F_BACnetRM_IsErrorSet:=TRUE;
IF stResult^.errorType = E_BACnet_ErrorType.eTypeAbort AND stResult^.abortReason = E_BACnet_AbortReason.eNoError THEN
	F_BACnetRM_IsErrorSet:=FALSE;
	RETURN;
END_IF
IF stResult^.errorType = E_BACnet_ErrorType.eTypeError AND stResult^.errorClass = E_BACnet_ErrorClass.eErrorClassNoError THEN
	F_BACnetRM_IsErrorSet:=FALSE;
	RETURN;
END_IF
IF stResult^.errorType = E_BACnet_ErrorType.eTypeReject AND stResult^.rejectCode = E_BACnet_RejectReason.eNoError THEN
	F_BACnetRM_IsErrorSet:=FALSE;
	RETURN;
END_IF

END_FUNCTION

// POUs/Helper/[internal]/String/F_BACnet_ChrStrExtLen
{attribute 'hide'} // [Workaround] Not hidden when lib is included
FUNCTION INTERNAL F_BACnet_ChrStrExtLen : UDINT
VAR
	pByte	: POINTER TO BYTE;
	nLen	: UDINT;
END_VAR
(*All VAR_IN_OUT variables have been moved to the end of the declaration due to compatibility reasons*)
VAR_IN_OUT
	stCharStringExt	: ST_BACnet_CharacterStringExt;
END_VAR

pByte := ADR(stCharStringExt);
nLen := SIZEOF(stCharStringExt);
(* check the string type *)
IF (nLen > 4 AND stCharStringExt.cookie = 0) THEN
	(* character string ext. *)
	IF (stCharStringExt.strLen <= SIZEOF(stCharStringExt.stringData)) THEN
		(* plausible string length given *)
		F_BACnet_ChrStrExtLen := stCharStringExt.strLen;
		RETURN;
	END_IF
	(* use sizeof, because string length isn't plausible *)
	nLen := SIZEOF(stCharStringExt.stringData);
	(* re-adjust pointer *)
	pByte := ADR(stCharStringExt.stringData);
END_IF
(* scan zero termination *)
F_BACnet_ChrStrExtLen := 0;
WHILE ((pByte^ <> 0) AND (F_BACnet_ChrStrExtLen < nLen)) DO
	pByte := pByte + 1;
	F_BACnet_ChrStrExtLen := F_BACnet_ChrStrExtLen + 1;
END_WHILE

END_FUNCTION

// POUs/Helper/[internal]/String/F_BACnet_DecodeUCS2
{attribute 'hide'} // [Workaround] Not hidden when lib is included
FUNCTION INTERNAL F_BACnet_DecodeUCS2 : UDINT (* result is the new character length of the string *)
VAR_INPUT
	pString		: POINTER TO WORD; (* pointer to UCS2 string beginning *)
	nString	: UDINT; (* byte size of string (use SIZEOF - don't use LEN) *)
END_VAR
VAR
	i		: UDINT;
	pResult	: POINTER TO BYTE;
	pBy		: POINTER TO WORD;
END_VAR

pResult	:= pString;
pBy		:= pString;
FOR i := 0 TO nString-1 DO
	pResult^ := F_BACnet_UCS2ToWin1252(pBy, TRUE);
	pBy := pBy + 2;
	(* end-of-string by character *)
	IF (pResult^ = 16#00) THEN
		EXIT;
	END_IF
	(* next character *)
	pResult := pResult + 1;
	(* end-of-string by length *)
	IF (pBy >= (pString + nString)) THEN
		EXIT;
	END_IF
END_FOR
pResult^ := 16#00;
F_BACnet_DecodeUCS2 := pResult - pString;

END_FUNCTION

// POUs/Helper/[internal]/String/F_BACnet_UCS2ToWin1252
{attribute 'hide'} // [Workaround] Not hidden when lib is included
FUNCTION INTERNAL F_BACnet_UCS2ToWin1252 : BYTE
VAR_INPUT
	pUCS2 :	POINTER TO WORD;
	bBE	: BOOL; (* byte-order big endian = TRUE *)
END_VAR
VAR
	pArr : POINTER TO ARRAY[0..1] OF BYTE;
	wUCS2: WORD;
END_VAR
VAR CONSTANT
	cRepl	: BYTE := 16#5F;
END_VAR

(*
	Windows-Codepages
874		Thai
932		Japanisch
936		Vereinfachtes Chinesisch
949		Koreanisch
950		Traditionelles Chinesisch
1250	Mitteleuropäisch
1251	Kyrillisch
1252	Westeuropäisch
1253	Griechisch
1254	Türkisch
1255	Hebräisch
1256	Arabisch
1257	Baltisch
1258	Vietnamesisch
*)
pArr := pUCS2;
IF bBE THEN
	wUCS2 := (pArr^[0] * 16#0100) + pArr^[1];
ELSE
	wUCS2 := pUCS2^;
END_IF
CASE wUCS2 OF
	16#178: 	F_BACnet_UCS2ToWin1252 := 16#9F;
	16#153: 	F_BACnet_UCS2ToWin1252 := 16#9C;
	16#152: 	F_BACnet_UCS2ToWin1252 := 16#8C;
	16#17E: 	F_BACnet_UCS2ToWin1252 := 16#9E;
	16#17D: 	F_BACnet_UCS2ToWin1252 := 16#8E;
	16#161: 	F_BACnet_UCS2ToWin1252 := 16#9A;
	16#160: 	F_BACnet_UCS2ToWin1252 := 16#8A;
	16#20AC: 	F_BACnet_UCS2ToWin1252 := 16#80;
	ELSE
		IF wUCS2 <= 16#FF THEN
			F_BACnet_UCS2ToWin1252 := WORD_TO_BYTE(wUCS2);
		ELSE
			F_BACnet_UCS2ToWin1252 := cRepl;
		END_IF
END_CASE

END_FUNCTION

// POUs/Helper/[internal]/String/F_BACnet_DecodeUCS4
{attribute 'hide'} // [Workaround] Not hidden when lib is included
FUNCTION INTERNAL F_BACnet_DecodeUCS4 : UDINT (* result is the new character length of the string *)
VAR_INPUT
	pString		: POINTER TO DWORD; (* pointer to UCS4 string beginning *)
	nString	: UDINT; (* byte size of string (use SIZEOF - don't use LEN) *)
END_VAR
VAR
	i		: UDINT;
	pResult	: POINTER TO BYTE;
	pBy		: POINTER TO WORD;
END_VAR

pResult	:= pString;
pBy		:= pString;
FOR i := 0 TO nString-1 DO
	(* byte order big endian *)
	pResult^ := F_BACnet_UCS2ToWin1252(pBy+2, TRUE);
	pBy := pBy + 4;
	(* end-of-string by character *)
	IF (pResult^ = 16#00) THEN
		EXIT;
	END_IF
	(* next character *)
	pResult := pResult + 1;
	(* end-of-string by length *)
	IF (pBy >= (pString + nString)) THEN
		EXIT;
	END_IF
END_FOR
pResult^ := 16#00;
F_BACnet_DecodeUCS4 := pResult - pString;

END_FUNCTION

// POUs/Helper/[internal]/String/F_BACnet_DecodeUTF8
{attribute 'hide'} // [Workaround] Not hidden when lib is included
FUNCTION INTERNAL F_BACnet_DecodeUTF8 : UDINT (* result is the new character length of the string *)
VAR_INPUT
	pString		: POINTER TO BYTE; (* pointer to UTF-8 string beginning *)
	nString	: UDINT; (* byte size of string (use SIZEOF - don't use LEN) *)
END_VAR
VAR
	i			: UDINT;
	pResult		: POINTER TO BYTE;
	pBy			: POINTER TO BYTE;
	pByArr		: POINTER TO ARRAY[0..3] OF BYTE;
END_VAR

pResult	:= pString;
pBy		:= pString;
FOR i := 0 TO nString-1 DO
	pByArr := pBy;
	IF (pByArr^[0] AND 16#F0) = 16#C0 THEN
		IF (pByArr^[1] AND 16#80) = 16#80 THEN
			pResult^ := F_BACnet_Utf8ToWin1252(pByArr, 2);
			pBy := pBy + 2;
		END_IF
	ELSIF (pByArr^[0] AND 16#F0) = 16#E0 THEN
		IF (pByArr^[1] AND 16#80) = 16#80 THEN
			IF (pByArr^[2] AND 16#80) = 16#80 THEN
				pResult^ := F_BACnet_Utf8ToWin1252(pByArr, 3);
				pBy := pBy + 3;
			END_IF
		END_IF
	ELSIF (pByArr^[0] AND 16#F0) = 16#F0 THEN
		IF (pByArr^[1] AND 16#80) = 16#80 THEN
			IF (pByArr^[2] AND 16#80) = 16#80 THEN
				IF (pByArr^[3] AND 16#80) = 16#80 THEN
					pResult^ := F_BACnet_Utf8ToWin1252(pByArr, 4);
					pBy := pBy + 4;
				END_IF
			END_IF
		END_IF
	ELSE
		(* ASCII character *)
		pResult^ := pBy^;
		pBy := pBy + 1;
	END_IF
	(* end-of-string by character *)
	IF (pResult^ = 16#00) THEN
		EXIT;
	END_IF
	(* next character *)
	pResult := pResult + 1;
	(* end-of-string by length *)
	IF (pBy >= (pString + nString)) THEN
		EXIT;
	END_IF
END_FOR
pResult^ := 16#00;
F_BACnet_DecodeUTF8 := pResult - pString;

END_FUNCTION

// POUs/Helper/[internal]/String/F_BACnet_Utf8ToWin1252
{attribute 'hide'} // [Workaround] Not hidden when lib is included
FUNCTION INTERNAL F_BACnet_Utf8ToWin1252 : BYTE
VAR_INPUT
	pUtf8	: POINTER TO BYTE;
	nUtf8	: UDINT; (* byte size of UTF8 character (1...6) *)
END_VAR
VAR
	pArr		: POINTER TO ARRAY[0..5] OF BYTE;
	pWord		: POINTER TO ARRAY[0..1] OF BYTE;
	wUCS2		: WORD;
END_VAR
VAR CONSTANT
	cRepl	: BYTE := 16#5F;
END_VAR

(*
	Windows-Codepages
874		Thai
932		Japanisch
936		Vereinfachtes Chinesisch
949		Koreanisch
950		Traditionelles Chinesisch
1250	Mitteleuropäisch
1251	Kyrillisch
1252	Westeuropäisch
1253	Griechisch
1254	Türkisch
1255	Hebräisch
1256	Arabisch
1257	Baltisch
1258	Vietnamesisch
*)
(* first step - convert to UCS2 *)
pArr := pUtf8;
IF (pArr^[0] <= 16#7F) THEN
	(* basic latin *)
	F_BACnet_Utf8ToWin1252 := pArr^[0];
	RETURN;
ELSIF (nUtf8 >= 2) THEN
	pWord := ADR(wUCS2);
	IF (pArr^[0] = 16#C2) THEN
		(* latin-1 supplement *)
		wUCS2 := pArr^[1];
	ELSIF (pArr^[0] = 16#C3) AND (pArr^[1] <= 16#BF) THEN
		(* latin-1 supplement *)
		wUCS2 := pArr^[1] + 16#40;
	ELSIF (pArr^[0] = 16#C4) AND (pArr^[1] >= 16#80) THEN
		(* latin extended-A *)
		pWord^[1] := 16#01;
		pWord^[0] := pArr^[1] - 16#80;
	ELSIF (pArr^[0] = 16#C5) AND (pArr^[1] >= 16#80) THEN
		(* latin extended-A *)
		pWord^[1] := 16#01;
		pWord^[0] := pArr^[1] - 16#40;
	ELSIF (pArr^[0] = 16#C6) AND (pArr^[1] >= 16#80) THEN
		(* latin extended-B *)
		pWord^[1] := 16#01;
		pWord^[0] := pArr^[1];
	ELSIF (pArr^[0] = 16#C7) AND (pArr^[1] <= 16#BF) THEN
		(* latin extended-B *)
		pWord^[1] := 16#01;
		pWord^[0] := pArr^[1] + 16#40;
	ELSIF (nUtf8 >= 3) THEN
		IF (pArr^[0] = 16#E2) AND (pArr^[1] = 16#82) THEN
			(* currency symbols *)
			pWord^[1] := 16#20;
			pWord^[0] := pArr^[2];
		ELSE
			(* unsupported *)
			F_BACnet_Utf8ToWin1252 := cRepl;
			RETURN;
		END_IF
	ELSE
		(* unsupported *)
		F_BACnet_Utf8ToWin1252 := cRepl;
		RETURN;
	END_IF
	(* convert UCS2 to Windows-1252 *)
	F_BACnet_Utf8ToWin1252 := F_BACnet_UCS2ToWin1252(pWord, FALSE);
	RETURN;
END_IF
(* unsupported *)
F_BACnet_Utf8ToWin1252 := cRepl;

END_FUNCTION

// POUs/Helper/[internal]/String/F_BACnet_EncodeUTF8
{attribute 'hide'} // [Workaround] Not hidden when lib is included
FUNCTION INTERNAL F_BACnet_EncodeUTF8 : UDINT (* actually byte length of the result utf-8 string (maybe longer than cbResult; means overflow) *)
VAR_INPUT
	pString		: POINTER TO BYTE; (* pointer to Win1252 string beginning *)
	nString	: UDINT; (* byte size of string (use SIZEOF - don't use LEN) *)
	pResult		: POINTER TO BYTE; (* pointer to result UTF-8 data area *)
	nResult	: UDINT; (* byte size of result (use SIZEOF - don't use LEN) *)
END_VAR

VAR
	pBy			: POINTER TO BYTE;
	pByArr		: POINTER TO ARRAY[0..3] OF BYTE;
	nCoded		: UINT;
	bOverflow	: BOOL;
END_VAR
(*All VAR_IN_OUT variables have been moved to the end of the declaration due to compatibility reasons*)
VAR_IN_OUT
	nResultLen	: UDINT; (* final resulting string length (<= nResult) *)
END_VAR

pBy			:= pString;
pByArr		:= pResult;
bOverflow	:= FALSE;
F_BACnet_EncodeUTF8 := 0;
nResultLen	:= 0;
(* loop over pString *)
WHILE pBy < (pString + nString) DO
	IF (pBy^ = 0) THEN EXIT; END_IF
	IF bOverflow OR (F_BACnet_EncodeUTF8 + 3 > nResult) THEN
		nCoded := F_BACnet_Win1252ToUtf8(nW1252:=pBy^, pUtf8:=pByArr, bEval:=TRUE);
		IF (NOT bOverflow) AND (F_BACnet_EncodeUTF8 + nCoded <= nResult) THEN
			nCoded := F_BACnet_Win1252ToUtf8(nW1252:=pBy^, pUtf8:=pByArr, bEval:=FALSE);
		ELSE
			bOverflow := TRUE;
		END_IF
	ELSE
		nCoded := F_BACnet_Win1252ToUtf8(nW1252:=pBy^, pUtf8:=pByArr, bEval:=FALSE);
	END_IF
	IF (NOT bOverflow) THEN
		pByArr := pByArr + UINT_TO_UDINT(nCoded);
		nResultLen := F_BACnet_EncodeUTF8 + nCoded;
	END_IF
	F_BACnet_EncodeUTF8 := F_BACnet_EncodeUTF8 + nCoded;
	pBy := pBy + 1;
END_WHILE
(* add zero termination if needed *)
IF (nResultLen < nResult) THEN
	pByArr^[0] := 16#00;
END_IF

END_FUNCTION

// POUs/Helper/[internal]/String/F_BACnet_Win1252ToUtf8
{attribute 'hide'} // [Workaround] Not hidden when lib is included
FUNCTION INTERNAL F_BACnet_Win1252ToUtf8 : UINT(0..3)
VAR_INPUT
	nW1252	: BYTE; (* Win1252 character *)
	pUtf8	: POINTER TO ARRAY[0..2] OF BYTE; (* pointer to target character buffer (utf-8) *)
	bEval	: BOOL; (* TRUE = only evaluate expected coding size (0..3 byte) - but don't write data *)
END_VAR
VAR
	pWord	: POINTER TO ARRAY[0..1] OF BYTE;
	wUCS2	: WORD;
END_VAR
VAR CONSTANT
	cRepl	: BYTE := 16#5F;
END_VAR

(*
	Windows-Codepages
874		Thai
932		Japanisch
936		Vereinfachtes Chinesisch
949		Koreanisch
950		Traditionelles Chinesisch
1250	Mitteleuropäisch
1251	Kyrillisch
1252	Westeuropäisch
1253	Griechisch
1254	Türkisch
1255	Hebräisch
1256	Arabisch
1257	Baltisch
1258	Vietnamesisch
*)
(* check pointer *)
IF (pUtf8 = 0) THEN
	(* null pointer *)
	F_BACnet_Win1252ToUtf8 := 0;
ELSIF (nW1252 <= 16#7F) THEN
	(* basic latin - 1 byte *)
	IF (NOT bEval) THEN
		pUtf8^[0] := nW1252;
	END_IF
	F_BACnet_Win1252ToUtf8 := 1;
ELSE
	(* convert to UCS-2 first *)
	wUCS2 := F_BACnet_Win1252ToUCS2(nW1252:=nW1252, bBE:=FALSE);
	pWord := ADR(wUCS2);
	(* convert used ranges *)
	IF (wUCS2 >= 16#80 AND wUCS2 <= 16#BF) THEN
		(* latin-1 supplement *)
		IF (NOT bEval) THEN
			pUtf8^[0] := 16#C2;
			pUtf8^[1] := pWord^[0];
		END_IF
		F_BACnet_Win1252ToUtf8 := 2;
	ELSIF (wUCS2 >= 16#C0 AND wUCS2 <= 16#FF) THEN
		(* latin-1 supplement *)
		IF (NOT bEval) THEN
			pUtf8^[0] := 16#C3;
			pUtf8^[1] := pWord^[0] - 16#40;
		END_IF
		F_BACnet_Win1252ToUtf8 := 2;
	ELSIF (wUCS2 >= 16#140 AND wUCS2 <= 16#17F) THEN
		(* latin extended A *)
		IF (NOT bEval) THEN
			pUtf8^[0] := 16#C5;
			pUtf8^[1] := pWord^[0] + 16#40;
		END_IF
		F_BACnet_Win1252ToUtf8 := 2;
	ELSIF (wUCS2 >= 16#20A0 AND wUCS2 <= 16#20BF) THEN
		(* currency symbols *)
		IF (NOT bEval) THEN
			pUtf8^[0] := 16#E2;
			pUtf8^[1] := 16#82;
			pUtf8^[2] := pWord^[0];
		END_IF
		F_BACnet_Win1252ToUtf8 := 3;
	ELSE
		(* unsupported *)
		IF (NOT bEval) THEN
			pUtf8^[0] := cRepl;
		END_IF
		F_BACnet_Win1252ToUtf8 := 1;
	END_IF
END_IF

END_FUNCTION

// POUs/Helper/[internal]/String/F_BACnet_Win1252ToUCS2
{attribute 'hide'} // [Workaround] Not hidden when lib is included
FUNCTION INTERNAL F_BACnet_Win1252ToUCS2 : WORD
VAR_INPUT
	nW1252 : BYTE;
	bBE	: BOOL; (* byte-order big endian = TRUE *)
END_VAR
VAR
	pArr : POINTER TO ARRAY[0..1] OF BYTE;
	nBuf : BYTE;
	wUCS2: WORD;
END_VAR

(*
	Windows-Codepages
874		Thai
932		Japanisch
936		Vereinfachtes Chinesisch
949		Koreanisch
950		Traditionelles Chinesisch
1250	Mitteleuropäisch
1251	Kyrillisch
1252	Westeuropäisch
1253	Griechisch
1254	Türkisch
1255	Hebräisch
1256	Arabisch
1257	Baltisch
1258	Vietnamesisch
*)
CASE nW1252 OF
	16#9F: wUCS2 := 16#178;
	16#9C: wUCS2 := 16#153;
	16#8C: wUCS2 := 16#152;
	16#9E: wUCS2 := 16#17E;
	16#8E: wUCS2 := 16#17D;
	16#9A: wUCS2 := 16#161;
	16#8A: wUCS2 := 16#160;
	16#80: wUCS2 := 16#20AC;
	ELSE
	wUCS2 := nW1252;
END_CASE
IF bBE THEN
	pArr := ADR(wUCS2);
	nBuf := pArr^[0];
	pArr^[0] := pArr^[1];
	pArr^[1] := nBuf;
END_IF
F_BACnet_Win1252ToUCS2 := wUCS2;

END_FUNCTION

// POUs/Helper/[internal]/String/F_BACnet_GetUsedStateText
{attribute 'hide'} // [Workaround] Not hidden when lib is included
FUNCTION INTERNAL F_BACnet_GetUsedStateText : UDINT
VAR_IN_OUT
	sArray				: ARRAY[*] OF T_BACnet_StateText;
END_VAR
VAR
	_nTemp				: DINT;
END_VAR

F_BACnet_GetUsedStateText := 0;

FOR _nTemp := LOWER_BOUND(sArray, 1) TO UPPER_BOUND(sArray, 1) DO
	IF LEN(sArray[_nTemp]) = 0 THEN
		EXIT;
	ELSE
		F_BACnet_GetUsedStateText := (F_BACnet_GetUsedStateText+1);
	END_IF
END_FOR

END_FUNCTION

// POUs/Helper/[internal]/String/F_BACnet_GetUsedUDINT
{attribute 'hide'} // [Workaround] Not hidden when lib is included
FUNCTION INTERNAL F_BACnet_GetUsedUDINT : UDINT
VAR_IN_OUT
	nArray				: ARRAY[*] OF UDINT;
END_VAR
VAR
	_nTemp				: DINT;
END_VAR

F_BACnet_GetUsedUDINT := 0;

FOR _nTemp := LOWER_BOUND(nArray, 1) TO UPPER_BOUND(nArray, 1) DO
	IF (nArray[_nTemp] = 0) THEN
		EXIT;
	ELSE
		F_BACnet_GetUsedUDINT := (F_BACnet_GetUsedUDINT+1);
	END_IF
END_FOR

END_FUNCTION

// POUs/Helper/[internal]/Validation-Functions/F_BACnet_IsObjIdentifierValid
{attribute 'hide'} // [Workaround] Not hidden when lib is included
FUNCTION INTERNAL F_BACnet_IsObjIdentifierValid : BOOL
VAR_INPUT
	tIdentifier		: T_BACnet_ObjectIdentifier;
END_VAR

F_BACnet_IsObjIdentifierValid := ((tIdentifier <> 0) AND (tIdentifier <> BACnet_Globals.nBACnetObjId_None));

END_FUNCTION

// POUs/Helper/[internal]/Validation-Functions/F_BACnet_IsPriorityValid
{attribute 'hide'} // [Workaround] Not hidden when lib is included
FUNCTION INTERNAL F_BACnet_IsPriorityValid : BOOL
VAR_INPUT
	ePriority		: E_BACnet_Priority;
END_VAR

F_BACnet_IsPriorityValid := ((E_BACnet_Priority.First <= ePriority) AND (ePriority <= E_BACnet_Priority.Last));

END_FUNCTION

// POUs/Helper/[internal]/Validation-Functions/F_BACnet_IsSchedBTypeValid
{attribute 'hide'} // [Workaround] Not hidden when lib is included
FUNCTION INTERNAL F_BACnet_IsSchedBTypeValid : BOOL
VAR_INPUT
	eType		: E_BACnet_SchedBType;
END_VAR

F_BACnet_IsSchedBTypeValid := ((E_BACnet_SchedBType.First <= eType) AND (eType <= E_BACnet_SchedBType.Last));

END_FUNCTION

// POUs/Helper/[internal]/F_BACnet_AlignedSize
{attribute 'hide'} // [Workaround] Not hidden when lib is included
FUNCTION INTERNAL F_BACnet_AlignedSize : DWORD
VAR_INPUT
	n	: DWORD;
END_VAR
VAR
END_VAR

F_BACnet_AlignedSize := (4*(((n)+3)/4));

END_FUNCTION

// POUs/Helper/[internal]/F_BACnet_AnalogPV
{attribute 'hide'} // [Workaround] Not hidden when lib is included
FUNCTION INTERNAL F_BACnet_AnalogPV : REAL
VAR_INPUT
	bEnable	: BOOL; (* TRUE = commit to stack, FALSE = do-nothing *)
	bNull	: BOOL; (* TRUE = clear priority, FALSE = write value from input *)
	fValue	: REAL;
END_VAR
VAR
	pres : POINTER TO DWORD;
END_VAR

IF (bEnable) THEN
	IF (bNull) THEN
		pres := ADR(F_BACnet_AnalogPV);
		pres^ := F_BACnet_RealNull(); 
	ELSE
		F_BACnet_AnalogPV := fValue;
	END_IF
ELSE
	F_BACnet_AnalogPV := F_BACnet_NAN();
END_IF

END_FUNCTION

// POUs/Helper/Real/F_BACnet_RealNull
FUNCTION F_BACnet_RealNull : DWORD
(* function that generates <not-a-number> real state *)

F_BACnet_RealNull:=16#7FFF0000;

END_FUNCTION

// POUs/Helper/Real/F_BACnet_NAN
FUNCTION F_BACnet_NAN : REAL
(* function that generates <not-a-number> real state *)
VAR
	res : POINTER TO DWORD;
END_VAR

res:=ADR(F_BACnet_NAN);
res^:=16#7FFFFFFF;

END_FUNCTION

// POUs/Helper/[internal]/F_BACnet_BitFieldBit
{attribute 'hide'} // [Workaround] Not hidden when lib is included
FUNCTION INTERNAL F_BACnet_BitFieldBit : WORD
VAR_INPUT
	bitNbr	:	INT;
END_VAR
VAR
END_VAR

F_BACnet_BitFieldBit := to_word((bitNbr/8) * 8 + (bitNbr MOD 8));

END_FUNCTION

// POUs/Helper/[internal]/F_BACnet_ChangeBitFieldBit
{attribute 'hide'} // [Workaround] Not hidden when lib is included
FUNCTION INTERNAL F_BACnet_ChangeBitFieldBit : DWORD
VAR_INPUT
	ptrData		: POINTER TO DWORD;
	bitNbr			: INT;
	Value		: BOOL;
END_VAR
VAR
END_VAR

IF (NOT Value) THEN
	ptrData^ := ptrData^ AND NOT (SHR(DWORD#16#00008000,F_BACnet_BitFieldBit(bitNbr)));
ELSE
	ptrData^ := ptrData^ OR (SHR(DWORD#16#00008000,F_BACnet_BitFieldBit(bitNbr)));
END_IF
F_BACnet_ChangeBitFieldBit := ptrData^;

END_FUNCTION

// POUs/Helper/[internal]/F_BACnet_EndOf
{attribute 'hide'} // [Workaround] Not hidden when lib is included
FUNCTION INTERNAL F_BACnet_EndOf : POINTER TO BYTE
VAR_INPUT
	 pPtr : POINTER TO BYTE;
	 nSize : DWORD;
END_VAR
VAR
END_VAR

F_BACnet_EndOf:=pPtr+nSize;

END_FUNCTION

// POUs/Helper/[internal]/F_BACnet_IsBitFieldBitSet
{attribute 'hide'} // [Workaround] Not hidden when lib is included
FUNCTION INTERNAL F_BACnet_IsBitFieldBitSet : BOOL
VAR_INPUT
	data	:	DWORD;
	bitNbr		:	INT;
END_VAR
VAR
END_VAR

F_BACnet_IsBitFieldBitSet:= (data AND (SHR(DWORD#16#00008000,F_BACnet_BitFieldBit(bitNbr)))) > 0;

END_FUNCTION

// POUs/Helper/[internal]/F_BACnet_IsBitFieldBitSetPtr
{attribute 'hide'} // [Workaround] Not hidden when lib is included
FUNCTION INTERNAL F_BACnet_IsBitFieldBitSetPtr : BOOL
VAR_INPUT
	pData	:	POINTER TO WORD;
	bitNbr	:	INT;
END_VAR
VAR
END_VAR

F_BACnet_IsBitFieldBitSetPtr:= ((pData^) AND (SHR(16#8000,F_BACnet_BitFieldBit(bitNbr)))) > 0;

END_FUNCTION

// POUs/Helper/[internal]/F_BACnet_NextListElem
{attribute 'hide'} // [Workaround] Not hidden when lib is included
FUNCTION INTERNAL F_BACnet_NextListElem : POINTER TO BYTE
VAR_INPUT
	 pPtr : POINTER TO BYTE;
	 nSize : DWORD;
END_VAR
VAR
END_VAR

IF nSize < 16#80000000 THEN
	F_BACnet_NextListElem:=0;
	RETURN;
END_IF
F_BACnet_NextListElem:=pPtr+F_BACnet_AlignedSize(nSize AND 16#7FFFFFFF)+8;

END_FUNCTION

// POUs/Helper/[internal]/F_BACnet_SetBitFieldBit
{attribute 'hide'} // [Workaround] Not hidden when lib is included
FUNCTION INTERNAL F_BACnet_SetBitFieldBit : DWORD
VAR_INPUT
	ptrData		:	POINTER TO DWORD;
	bitNbr			:	INT;
END_VAR
VAR
END_VAR

ptrData^ := ptrData^ OR (SHR(DWORD#16#00008000, F_BACnet_BitFieldBit(bitNbr)));
F_BACnet_SetBitFieldBit := ptrData^;

END_FUNCTION

// POUs/Helper/[internal]/F_BACnet_SysTimeDiff
{attribute 'hide'} // [Workaround] Not hidden when lib is included
FUNCTION INTERNAL F_BACnet_SysTimeDiff : REAL
VAR_INPUT
	In1, In2 : T_LARGE_INTEGER;
END_VAR

F_BACnet_SysTimeDiff := LREAL_TO_REAL(INT64_TO_LREAL(Int64Sub64(In1, In2)) / 10000000.0); (* [s] *)

END_FUNCTION

// POUs/Helper/[internal]/F_BACnet_UnSetBitFieldBit
{attribute 'hide'} // [Workaround] Not hidden when lib is included
FUNCTION INTERNAL F_BACnet_UnSetBitFieldBit : DWORD
VAR_INPUT
	ptrData		:	POINTER TO DWORD;
	bitNbr			:	INT;
END_VAR
VAR
END_VAR

ptrData^ := ptrData^ AND NOT (SHR(DWORD#16#00008000,F_BACnet_BitFieldBit(bitNbr)));
F_BACnet_UnSetBitFieldBit := ptrData^;

END_FUNCTION

// POUs/Helper/Flags/F_BACnet_EventEnable
FUNCTION F_BACnet_EventEnable : UINT
VAR_INPUT
	stEvtEn       : ST_BA_EventTransitions;
END_VAR
VAR
	nEvtEnToFlt     : UINT;
	nEvtEnToNmal    : UINT;
	nEvtEnToOffnmal : UINT;
	nEvtEnNo        : UINT;
END_VAR

(*=============================================*)
(*EventEnable*)
IF	stEvtEn.bToFault
THEN
	nEvtEnToFlt := 16#4000;
ELSE
	nEvtEnToFlt := 16#0;
END_IF

IF	stEvtEn.bToNormal
THEN
	nEvtEnToNmal := 16#2000;
ELSE
	nEvtEnToNmal := 16#0;
END_IF

IF	stEvtEn.bToOffnormal
THEN
	nEvtEnToOffnmal := 16#8000;
ELSE
	nEvtEnToOffnmal := 16#0;
END_IF

nEvtEnNo := 5;

F_BACnet_EventEnable := nEvtEnNo + nEvtEnToFlt + nEvtEnToNmal + nEvtEnToOffnmal;
(*=============================================*)

END_FUNCTION

// POUs/Helper/Flags/F_BACnet_EventTransitionFlags
FUNCTION F_BACnet_EventTransitionFlags : ST_BA_EventTransitions
VAR_INPUT
	data	: WORD;
END_VAR
VAR
END_VAR

F_BACnet_EventTransitionFlags.bToNormal := F_BACnet_IsBitFieldBitSet(data, E_BACnet_EventTransitionBits.eToNormal);
F_BACnet_EventTransitionFlags.bToOffnormal := F_BACnet_IsBitFieldBitSet(data, E_BACnet_EventTransitionBits.eToOffnormal);
F_BACnet_EventTransitionFlags.bToFault := F_BACnet_IsBitFieldBitSet(data, E_BACnet_EventTransitionBits.eToFault);

END_FUNCTION

// POUs/Helper/Flags/F_BACnet_GetEventTransFlagsData
FUNCTION F_BACnet_GetEventTransFlagsData : WORD
VAR_INPUT
	Flags	: ST_BA_EventTransitions;
END_VAR
VAR
END_VAR

F_BACnet_GetEventTransFlagsData := 16#0005;
IF Flags.bToNormal THEN
	F_BACnet_GetEventTransFlagsData := DWORD_TO_WORD(F_BACnet_SetBitFieldBit(ptrData:=ADR(F_BACnet_GetEventTransFlagsData), bitNbr:=E_BACnet_EventTransitionBits.eToNormal));
END_IF
IF Flags.bToOffnormal THEN
	F_BACnet_GetEventTransFlagsData := DWORD_TO_WORD(F_BACnet_SetBitFieldBit(ptrData:=ADR(F_BACnet_GetEventTransFlagsData), bitNbr:=E_BACnet_EventTransitionBits.eToOffnormal));
END_IF
IF Flags.bToFault THEN
	F_BACnet_GetEventTransFlagsData := DWORD_TO_WORD(F_BACnet_SetBitFieldBit(ptrData:=ADR(F_BACnet_GetEventTransFlagsData), bitNbr:=E_BACnet_EventTransitionBits.eToFault));
END_IF

END_FUNCTION

// POUs/Helper/Flags/F_BACnet_GetLimitEnFlagsData
FUNCTION F_BACnet_GetLimitEnFlagsData : WORD
VAR_INPUT
	Flags	: ST_BACnet_LimitEnable;
END_VAR
VAR
END_VAR

F_BACnet_GetLimitEnFlagsData := 16#0006;
IF Flags.highLimitEnable THEN
	F_BACnet_GetLimitEnFlagsData := DWORD_TO_WORD(F_BACnet_SetBitFieldBit(ptrData:=ADR(F_BACnet_GetLimitEnFlagsData), bitNbr:=E_BACnet_LimitEnableBits.eHighLimit));
END_IF
IF Flags.lowLimitEnable THEN
	F_BACnet_GetLimitEnFlagsData := DWORD_TO_WORD(F_BACnet_SetBitFieldBit(ptrData:=ADR(F_BACnet_GetLimitEnFlagsData), bitNbr:=E_BACnet_LimitEnableBits.eLowLimit));
END_IF

END_FUNCTION

// POUs/Helper/Flags/F_BACnet_GetStatusFlagsData
FUNCTION F_BACnet_GetStatusFlagsData : WORD
VAR_INPUT
	Flags : ST_BA_StatusFlags;
END_VAR

F_BACnet_GetStatusFlagsData	:= 16#0004;
IF Flags.bInAlarm THEN
	F_BACnet_GetStatusFlagsData := DWORD_TO_WORD(F_BACnet_SetBitFieldBit(ptrData:=ADR(F_BACnet_GetStatusFlagsData), bitNbr:=E_BACnet_StatusFlags.eInAlarm));
END_IF
IF Flags.bFault THEN
	F_BACnet_GetStatusFlagsData := DWORD_TO_WORD(F_BACnet_SetBitFieldBit(ptrData:=ADR(F_BACnet_GetStatusFlagsData), bitNbr:=E_BACnet_StatusFlags.eFault));
END_IF
IF Flags.bOverridden THEN
	F_BACnet_GetStatusFlagsData := DWORD_TO_WORD(F_BACnet_SetBitFieldBit(ptrData:=ADR(F_BACnet_GetStatusFlagsData), bitNbr:=E_BACnet_StatusFlags.eOverridden));
END_IF
IF Flags.bOutOfService THEN
	F_BACnet_GetStatusFlagsData := DWORD_TO_WORD(F_BACnet_SetBitFieldBit(ptrData:=ADR(F_BACnet_GetStatusFlagsData), bitNbr:=E_BACnet_StatusFlags.eOutOfService));
END_IF

END_FUNCTION

// POUs/Helper/Flags/F_BACnet_LimitEnable
FUNCTION F_BACnet_LimitEnable : UINT
VAR_INPUT
	stLimEn         : ST_BACnet_LimitEnable;
END_VAR
VAR
	nHiLimEn     : UINT;
	nLowLimEn    : UINT;
	nLimEnNo     : UINT;
END_VAR

(*=============================================*)
IF	stLimEn.highLimitEnable
THEN
	nHiLimEn := 16#4000;
ELSE
	nHiLimEn := 16#0;
END_IF


IF	stLimEn.lowLimitEnable
THEN
	nLowLimEn := 16#8000;
ELSE
	nLowLimEn := 16#0;
END_IF

nLimEnNo := 16#6;

F_BACnet_LimitEnable := nLimEnNo + nHiLimEn + nLowLimEn;
(*=============================================*)

END_FUNCTION

// POUs/Helper/Flags/F_BACnet_LimitEnableFlags
FUNCTION F_BACnet_LimitEnableFlags : ST_BACnet_LimitEnable
VAR_INPUT
	data	: WORD;
END_VAR
VAR
END_VAR

F_BACnet_LimitEnableFlags.highLimitEnable := F_BACnet_IsBitFieldBitSet( data:=data, bitNbr:=E_BACnet_LimitEnableBits.eHighLimit);
F_BACnet_LimitEnableFlags.lowLimitEnable := F_BACnet_IsBitFieldBitSet( data:=data, bitNbr:=E_BACnet_LimitEnableBits.eLowLimit);

END_FUNCTION

// POUs/Helper/Flags/F_BACnet_StatusFlags
FUNCTION F_BACnet_StatusFlags : ST_BA_StatusFlags
VAR_INPUT
	data	: WORD;
END_VAR
VAR
END_VAR

F_BACnet_StatusFlags.bInAlarm:= F_BACnet_IsBitFieldBitSet( data:=data, bitNbr:=E_BACnet_StatusFlags.eInAlarm);
F_BACnet_StatusFlags.bFault:= F_BACnet_IsBitFieldBitSet( data:=data, bitNbr:=E_BACnet_StatusFlags.eFault);
F_BACnet_StatusFlags.bOverridden:= F_BACnet_IsBitFieldBitSet( data:=data, bitNbr:=E_BACnet_StatusFlags.eOverridden);
F_BACnet_StatusFlags.bOutOfService:= F_BACnet_IsBitFieldBitSet( data:=data, bitNbr:=E_BACnet_StatusFlags.eOutOfService);

END_FUNCTION

// POUs/Helper/MultiState/F_BACnet_EnMultiStatePV
FUNCTION F_BACnet_EnMultiStatePV : UDINT
VAR_INPUT
	bEnable			: BOOL;
	nValue			: UDINT;
END_VAR

IF (bEnable) THEN
	F_BACnet_EnMultiStatePV := MAX(nValue, E_BACnet_MultistateVal.eMin);
ELSE
	F_BACnet_EnMultiStatePV := E_BACnet_MultistateVal.eNull;
END_IF

END_FUNCTION

// POUs/Helper/MultiState/F_BACnet_MultiStatePV
FUNCTION F_BACnet_MultiStatePV : UDINT
VAR_INPUT
	bEnable						: BOOL; (* TRUE = commit to stack, FALSE = do-nothing *)
	bNull						: BOOL; (* TRUE = clear priority, FALSE = write number from state input *)
	nState						: UDINT; (* multi-state [1..max-number-of-states] *)
END_VAR

IF (bEnable) THEN
	IF (bNull) THEN
		F_BACnet_MultiStatePV := E_BACnet_MultistateVal.eNull;
	ELSE
		F_BACnet_MultiStatePV := MAX(nState, E_BACnet_MultistateVal.eMin);
	END_IF
ELSE
	F_BACnet_MultiStatePV := E_BACnet_MultistateVal.eNothing;
END_IF

END_FUNCTION

// POUs/Helper/NC/F_BACnet_DeviceRecipient
// Returns an initialized recipient structure.
FUNCTION F_BACnet_DeviceRecipient : ST_BACnet_Recipient
VAR_INPUT
	nDeviceInstance		: UDINT			:= 16#003FFFFF;
END_VAR

F_BACnet_DeviceRecipient.eRecipientChoice := E_BACnet_RecipientChoice.eDevice;
F_BACnet_DeviceRecipient.stEntry.nDeviceInstance := F_BACnet_GetObjId(E_BACnetObjType.ObjDevice,nDeviceInstance);

END_FUNCTION

// POUs/Helper/F_BACnet_GetObjId
FUNCTION F_BACnet_GetObjId : T_BACnet_ObjectIdentifier
VAR_INPUT
	eObjectType		: E_BACnetObjType;
	nObjectInstance	: UDINT;
END_VAR
VAR
END_VAR

F_BACnet_GetObjId := F_BACnet_GetObjInstance(nObjectInstance) + SHL(INT_TO_UDINT(eObjectType), 22);

END_FUNCTION

// POUs/Helper/F_BACnet_GetObjInstance
FUNCTION F_BACnet_GetObjInstance : UDINT
VAR_INPUT
	nObjectId : DWORD;
END_VAR
VAR
END_VAR

F_BACnet_GetObjInstance := nObjectId AND 16#003FFFFF;

END_FUNCTION

// POUs/Helper/NC/F_BACnet_EthernetRecipient
// Returns an initialized recipient structure.
FUNCTION F_BACnet_EthernetRecipient : ST_BACnet_Recipient
VAR_INPUT
	nIPAddress1		: BYTE;
	nIPAddress2		: BYTE;
	nIPAddress3		: BYTE;
	nIPAddress4		: BYTE;
	nPort			: UINT;
	nNetworkNr		: UINT;
END_VAR
VAR
	_nPort			: POINTER TO ARRAY[0 .. 1] OF BYTE := ADR(nPort);
END_VAR

F_BACnet_EthernetRecipient.eRecipientChoice := E_BACnet_RecipientChoice.eAddress;
F_BACnet_EthernetRecipient.stEntry.stNetAddr.eChoice := E_BACnet_AddressChoice.eEthernet;
F_BACnet_EthernetRecipient.stEntry.stNetAddr.nNetworkNr := nNetworkNr;
F_BACnet_EthernetRecipient.stEntry.stNetAddr.eAddress[0] := nIPAddress1;
F_BACnet_EthernetRecipient.stEntry.stNetAddr.eAddress[1] := nIPAddress2;
F_BACnet_EthernetRecipient.stEntry.stNetAddr.eAddress[2] := nIPAddress3;
F_BACnet_EthernetRecipient.stEntry.stNetAddr.eAddress[3] := nIPAddress4;

// Swap Port-Bytes:
F_BACnet_EthernetRecipient.stEntry.stNetAddr.eAddress[4] := _nPort^[1];
F_BACnet_EthernetRecipient.stEntry.stNetAddr.eAddress[5] := _nPort^[0];

END_FUNCTION

// POUs/Helper/NC/F_BACnet_EthernetRecipientEx
// Returns an initialized recipient structure.
FUNCTION F_BACnet_EthernetRecipientEx : ST_BACnet_Recipient
VAR_INPUT
	tIPAddress		: T_IPv4AddrArr;
	nPort			: UINT;
	nNetworkNr		: UINT;
END_VAR

F_BACnet_EthernetRecipientEx := F_BACnet_EthernetRecipient(tIPAddress[0], tIPAddress[1], tIPAddress[2], tIPAddress[3], nPort, nNetworkNr);

END_FUNCTION

// POUs/Helper/Real/F_BACnet_EnRealPV
FUNCTION F_BACnet_EnRealPV : DWORD
VAR_INPUT
	bEnable	: BOOL;
	fValue	: REAL;
END_VAR
VAR
	pDword : POINTER TO DWORD;
END_VAR

IF (bEnable) THEN
	pDword := ADR(fValue);
	F_BACnet_EnRealPV := pDword^;
ELSE
	F_BACnet_EnRealPV := F_BACnet_RealNull();
END_IF

END_FUNCTION

// POUs/Helper/Real/F_BACnet_IsFinite
FUNCTION F_BACnet_IsFinite : BOOL
VAR_INPUT
	fValue		: REAL;
END_VAR
VAR
	fArg		: T_Arg;
END_VAR

fArg.cbLen := SIZEOF(fValue);
fArg.eType := ARGTYPE_REAL;
fArg.pData := ADR(fValue);
F_BACnet_IsFinite := IsFinite(fArg);

END_FUNCTION

// POUs/Helper/Real/F_BACnet_RealEQ
FUNCTION F_BACnet_RealEQ : BOOL
VAR_INPUT
	fIn1	: REAL;
	fIn2	: REAL;
END_VAR
VAR
END_VAR

IF (F_BACnet_IsFinite(fIn1) <> F_BACnet_IsFinite(fIn2)) THEN
	F_BACnet_RealEQ := FALSE;
	RETURN;
END_IF
IF F_BACnet_IsFinite(fIn1) THEN
	IF (fIn1 <> fIn2) THEN
		F_BACnet_RealEQ := FALSE;
		RETURN;
	END_IF
END_IF
F_BACnet_RealEQ := TRUE;

END_FUNCTION

// POUs/Helper/Real/F_BACnet_RealGE
FUNCTION F_BACnet_RealGE : BOOL
VAR_INPUT
	fIn1	: REAL;
	fIn2	: REAL;
END_VAR
VAR
END_VAR

IF NOT (F_BACnet_IsFinite(fIn1) OR F_BACnet_IsFinite(fIn2)) THEN
	F_BACnet_RealGE := FALSE;
	RETURN;
END_IF
F_BACnet_RealGE := (fIn1 >= fIn2);

END_FUNCTION

// POUs/Helper/Real/F_BACnet_RealGT
FUNCTION F_BACnet_RealGT : BOOL
VAR_INPUT
	fIn1	: REAL;
	fIn2	: REAL;
END_VAR
VAR
END_VAR

IF NOT (F_BACnet_IsFinite(fIn1) OR F_BACnet_IsFinite(fIn2)) THEN
	F_BACnet_RealGT := FALSE;
	RETURN;
END_IF
F_BACnet_RealGT := (fIn1 > fIn2);

END_FUNCTION

// POUs/Helper/Real/F_BACnet_RealLE
FUNCTION F_BACnet_RealLE : BOOL
VAR_INPUT
	fIn1	: REAL;
	fIn2	: REAL;
END_VAR
VAR
END_VAR

IF NOT (F_BACnet_IsFinite(fIn1) OR F_BACnet_IsFinite(fIn2)) THEN
	F_BACnet_RealLE := FALSE;
	RETURN;
END_IF
F_BACnet_RealLE := (fIn1 <= fIn2);

END_FUNCTION

// POUs/Helper/Real/F_BACnet_RealLT
FUNCTION F_BACnet_RealLT : BOOL
VAR_INPUT
	fIn1	: REAL;
	fIn2	: REAL;
END_VAR
VAR
END_VAR

IF NOT (F_BACnet_IsFinite(fIn1) OR F_BACnet_IsFinite(fIn2)) THEN
	F_BACnet_RealLT := FALSE;
	RETURN;
END_IF
F_BACnet_RealLT := (fIn1 < fIn2);

END_FUNCTION

// POUs/Helper/Real/F_BACnet_RealNothing
FUNCTION F_BACnet_RealNothing : DWORD

F_BACnet_RealNothing:=16#7FFFFFFF;

END_FUNCTION

// POUs/Helper/Real/F_BACnet_RealPV
FUNCTION F_BACnet_RealPV : DWORD
VAR_INPUT
	bEnable	: BOOL; (* TRUE = commit to stack, FALSE = do-nothing *)
	bNull	: BOOL; (* TRUE = clear priority, FALSE = write value from input *)
	fValue	: REAL;
END_VAR
VAR
	pDword : POINTER TO DWORD;
END_VAR

IF (bEnable) THEN
	IF (bNull) THEN
		F_BACnet_RealPV := F_BACnet_RealNull();
	ELSE
		pDword := ADR(fValue);
		F_BACnet_RealPV := pDword^;
	END_IF
ELSE
	F_BACnet_RealPV := F_BACnet_RealNothing();
END_IF

END_FUNCTION

// POUs/Helper/Real/F_BACnet_RealToStr
FUNCTION F_BACnet_RealToStr : STRING
VAR_INPUT
	pValue	: POINTER TO REAL;
END_VAR
VAR
	fArg	: T_Arg;
	pDWORD	: POINTER TO DWORD;
END_VAR

IF (pValue <> 0) THEN
	fArg.cbLen := 4;
	fArg.eType := ARGTYPE_REAL;
	fArg.pData := pValue;
	pDWORD := pValue;
	IF IsFinite(fArg) THEN
		F_BACnet_RealToStr := REAL_TO_STRING(pValue^);
	ELSE
		IF (pDWORD^ = 16#7FFF0000) THEN
			F_BACnet_RealToStr := '#NULL';
		ELSIF (pDWORD^ AND 16#80000000) = 16#80000000 THEN
			F_BACnet_RealToStr := '-#QNAN';
		ELSE
			F_BACnet_RealToStr := '#QNAN';
		END_IF
	END_IF
END_IF

END_FUNCTION

// POUs/Helper/Scheduler/Calendar/F_BACnet_SchedCalendar
// Returns an initialized analog weekly scheduler.
FUNCTION F_BACnet_SchedCalendar : T_BACnet_SchedCalendar
VAR_INPUT
	iRefCalendar1	: I_BACnet_Cal	:= 0;
	iRefCalendar2	: I_BACnet_Cal	:= 0;
	iRefCalendar3	: I_BACnet_Cal	:= 0;
END_VAR
VAR
	nIndex			: INT;
END_VAR

F_BACnet_SchedCalendar[1].iRefCalendar := iRefCalendar1;

nIndex := 2;
IF (BACnet_Param.nSched_CalendarCount >= nIndex) THEN
	F_BACnet_SchedCalendar[nIndex].iRefCalendar := iRefCalendar2;
END_IF

nIndex := 3;
IF (BACnet_Param.nSched_CalendarCount >= nIndex) THEN
	F_BACnet_SchedCalendar[nIndex].iRefCalendar := iRefCalendar3;
END_IF

END_FUNCTION

// POUs/Helper/Scheduler/Exception/F_BACnet_SchedEntry1xA
// Returns an initialized analog weekly scheduler.
FUNCTION F_BACnet_SchedEntry1xA : T_BACnet_SchedExceptionEntryList
VAR_INPUT
	tEntry1Time		: TIME;
	fEntry1Value	: REAL;
END_VAR

F_BA_SetSchedulerEntry(F_BACnet_SchedEntry1xA[1], tEntry1Time, F_BA_RVal(fEntry1Value));

END_FUNCTION

// POUs/Helper/Scheduler/Exception/F_BACnet_SchedEntry1xB
// Returns an initialized binary weekly scheduler.
FUNCTION F_BACnet_SchedEntry1xB : T_BACnet_SchedExceptionEntryList
VAR_INPUT
	tEntry1Time		: TIME;
	bEntry1Value	: BOOL;
END_VAR

F_BA_SetSchedulerEntry(F_BACnet_SchedEntry1xB[1], tEntry1Time, F_BA_BVal(bEntry1Value));

END_FUNCTION

// POUs/Helper/Scheduler/Exception/F_BACnet_SchedEntry1xM
// Returns an initialized multistate weekly scheduler.
FUNCTION F_BACnet_SchedEntry1xM : T_BACnet_SchedExceptionEntryList
VAR_INPUT
	tEntry1Time		: TIME;
	nEntry1Value	: UDINT;
END_VAR

F_BA_SetSchedulerEntry(F_BACnet_SchedEntry1xM[1], tEntry1Time, F_BA_UDIVal(nEntry1Value));

END_FUNCTION

// POUs/Helper/Scheduler/Exception/F_BACnet_SchedEntry3xA
// Returns an initialized analog weekly scheduler.
FUNCTION F_BACnet_SchedEntry3xA : T_BACnet_SchedExceptionEntryList
VAR_INPUT
	tEntry1Time		: TIME;
	fEntry1Value	: REAL;
	tEntry2Time		: TIME;
	fEntry2Value	: REAL;
	tEntry3Time		: TIME;
	fEntry3Value	: REAL;
END_VAR

F_BA_SetSchedulerEntry(F_BACnet_SchedEntry3xA[1], tEntry1Time, F_BA_RVal(fEntry1Value));
F_BA_SetSchedulerEntry(F_BACnet_SchedEntry3xA[2], tEntry2Time, F_BA_RVal(fEntry2Value));
F_BA_SetSchedulerEntry(F_BACnet_SchedEntry3xA[3], tEntry3Time, F_BA_RVal(fEntry3Value));

END_FUNCTION

// POUs/Helper/Scheduler/Exception/F_BACnet_SchedEntry3xB
// Returns an initialized binary weekly scheduler.
FUNCTION F_BACnet_SchedEntry3xB : T_BACnet_SchedExceptionEntryList
VAR_INPUT
	tEntry1Time		: TIME;
	bEntry1Value	: BOOL;
	tEntry2Time		: TIME;
	bEntry2Value	: BOOL;
	tEntry3Time		: TIME;
	bEntry3Value	: BOOL;
END_VAR

F_BA_SetSchedulerEntry(F_BACnet_SchedEntry3xB[1], tEntry1Time, F_BA_BVal(bEntry1Value));
F_BA_SetSchedulerEntry(F_BACnet_SchedEntry3xB[2], tEntry2Time, F_BA_BVal(bEntry2Value));
F_BA_SetSchedulerEntry(F_BACnet_SchedEntry3xB[3], tEntry3Time, F_BA_BVal(bEntry3Value));

END_FUNCTION

// POUs/Helper/Scheduler/Exception/F_BACnet_SchedEntry3xM
// Returns an initialized multistate weekly scheduler.
FUNCTION F_BACnet_SchedEntry3xM : T_BACnet_SchedExceptionEntryList
VAR_INPUT
	tEntry1Time		: TIME;
	nEntry1Value	: UDINT;
	tEntry2Time		: TIME;
	nEntry2Value	: UDINT;
	tEntry3Time		: TIME;
	nEntry3Value	: UDINT;
END_VAR

F_BA_SetSchedulerEntry(F_BACnet_SchedEntry3xM[1], tEntry1Time, F_BA_UDIVal(nEntry1Value));
F_BA_SetSchedulerEntry(F_BACnet_SchedEntry3xM[2], tEntry2Time, F_BA_UDIVal(nEntry2Value));
F_BA_SetSchedulerEntry(F_BACnet_SchedEntry3xM[3], tEntry3Time, F_BA_UDIVal(nEntry3Value));

END_FUNCTION

// POUs/Helper/Scheduler/Exception/F_BACnet_SchedEntry5xA
// Returns an initialized analog weekly scheduler.
FUNCTION F_BACnet_SchedEntry5xA : T_BACnet_SchedExceptionEntryList
VAR_INPUT
	tEntry1Time		: TIME;
	fEntry1Value	: REAL;
	tEntry2Time		: TIME;
	fEntry2Value	: REAL;
	tEntry3Time		: TIME;
	fEntry3Value	: REAL;
	tEntry4Time		: TIME;
	fEntry4Value	: REAL;
	tEntry5Time		: TIME;
	fEntry5Value	: REAL;
END_VAR

F_BA_SetSchedulerEntry(F_BACnet_SchedEntry5xA[1], tEntry1Time, F_BA_RVal(fEntry1Value));
F_BA_SetSchedulerEntry(F_BACnet_SchedEntry5xA[2], tEntry2Time, F_BA_RVal(fEntry2Value));
F_BA_SetSchedulerEntry(F_BACnet_SchedEntry5xA[3], tEntry3Time, F_BA_RVal(fEntry3Value));
F_BA_SetSchedulerEntry(F_BACnet_SchedEntry5xA[4], tEntry4Time, F_BA_RVal(fEntry4Value));
F_BA_SetSchedulerEntry(F_BACnet_SchedEntry5xA[5], tEntry5Time, F_BA_RVal(fEntry5Value));

END_FUNCTION

// POUs/Helper/Scheduler/Exception/F_BACnet_SchedEntry5xB
// Returns an initialized binary weekly scheduler.
FUNCTION F_BACnet_SchedEntry5xB : T_BACnet_SchedExceptionEntryList
VAR_INPUT
	tEntry1Time		: TIME;
	bEntry1Value	: BOOL;
	tEntry2Time		: TIME;
	bEntry2Value	: BOOL;
	tEntry3Time		: TIME;
	bEntry3Value	: BOOL;
	tEntry4Time		: TIME;
	bEntry4Value	: BOOL;
	tEntry5Time		: TIME;
	bEntry5Value	: BOOL;
END_VAR

F_BA_SetSchedulerEntry(F_BACnet_SchedEntry5xB[1], tEntry1Time, F_BA_BVal(bEntry1Value));
F_BA_SetSchedulerEntry(F_BACnet_SchedEntry5xB[2], tEntry2Time, F_BA_BVal(bEntry2Value));
F_BA_SetSchedulerEntry(F_BACnet_SchedEntry5xB[3], tEntry3Time, F_BA_BVal(bEntry3Value));
F_BA_SetSchedulerEntry(F_BACnet_SchedEntry5xB[4], tEntry4Time, F_BA_BVal(bEntry4Value));
F_BA_SetSchedulerEntry(F_BACnet_SchedEntry5xB[5], tEntry5Time, F_BA_BVal(bEntry5Value));

END_FUNCTION

// POUs/Helper/Scheduler/Exception/F_BACnet_SchedEntry5xM
// Returns an initialized multistate weekly scheduler.
FUNCTION F_BACnet_SchedEntry5xM : T_BACnet_SchedExceptionEntryList
VAR_INPUT
	tEntry1Time		: TIME;
	nEntry1Value	: UDINT;
	tEntry2Time		: TIME;
	nEntry2Value	: UDINT;
	tEntry3Time		: TIME;
	nEntry3Value	: UDINT;
	tEntry4Time		: TIME;
	nEntry4Value	: UDINT;
	tEntry5Time		: TIME;
	nEntry5Value	: UDINT;
END_VAR

F_BA_SetSchedulerEntry(F_BACnet_SchedEntry5xM[1], tEntry1Time, F_BA_UDIVal(nEntry1Value));
F_BA_SetSchedulerEntry(F_BACnet_SchedEntry5xM[2], tEntry2Time, F_BA_UDIVal(nEntry2Value));
F_BA_SetSchedulerEntry(F_BACnet_SchedEntry5xM[3], tEntry3Time, F_BA_UDIVal(nEntry3Value));
F_BA_SetSchedulerEntry(F_BACnet_SchedEntry5xM[4], tEntry4Time, F_BA_UDIVal(nEntry4Value));
F_BA_SetSchedulerEntry(F_BACnet_SchedEntry5xM[5], tEntry5Time, F_BA_UDIVal(nEntry5Value));

END_FUNCTION

// POUs/Helper/Scheduler/Weekly/F_BACnet_SchedWeekly1xA
// Returns an initialized analog weekly scheduler.
FUNCTION F_BACnet_SchedWeekly1xA : T_BACnet_SchedWeek
VAR_INPUT
	eDayFrom		: E_BA_Weekday		:= E_BA_Weekday.eMonday;
	eDayTo			: E_BA_Weekday		:= E_BA_Weekday.eSunday;
	
	tEntry1Time		: TIME;
	fEntry1Value	: REAL;
END_VAR

F_BA_SetWeekdays(F_BACnet_SchedWeekly1xA, eDayFrom, eDayTo, 1, tEntry1Time, F_BA_RVal(fEntry1Value));

END_FUNCTION

// POUs/Helper/Scheduler/Weekly/F_BACnet_SchedWeekly1xB
// Returns an initialized binary weekly scheduler.
FUNCTION F_BACnet_SchedWeekly1xB : T_BACnet_SchedWeek
VAR_INPUT
	eDayFrom		: E_BA_Weekday		:= E_BA_Weekday.eMonday;
	eDayTo			: E_BA_Weekday		:= E_BA_Weekday.eSunday;
	
	tEntry1Time		: TIME;
	bEntry1Value	: BOOL;
END_VAR

F_BA_SetWeekdays(F_BACnet_SchedWeekly1xB, eDayFrom, eDayTo, 1, tEntry1Time, F_BA_BVal(bEntry1Value));

END_FUNCTION

// POUs/Helper/Scheduler/Weekly/F_BACnet_SchedWeekly1xM
// Returns an initialized multistate weekly scheduler.
FUNCTION F_BACnet_SchedWeekly1xM : T_BACnet_SchedWeek
VAR_INPUT
	eDayFrom		: E_BA_Weekday		:= E_BA_Weekday.eMonday;
	eDayTo			: E_BA_Weekday		:= E_BA_Weekday.eSunday;
	
	tEntry1Time		: TIME;
	nEntry1Value	: UDINT;
END_VAR

F_BA_SetWeekdays(F_BACnet_SchedWeekly1xM, eDayFrom, eDayTo, 1, tEntry1Time, F_BA_UDIVal(nEntry1Value));

END_FUNCTION

// POUs/Helper/Scheduler/Weekly/F_BACnet_SchedWeekly3xA
// Returns an initialized analog weekly scheduler.
FUNCTION F_BACnet_SchedWeekly3xA : T_BACnet_SchedWeek
VAR_INPUT
	eDayFrom		: E_BA_Weekday		:= E_BA_Weekday.eMonday;
	eDayTo			: E_BA_Weekday		:= E_BA_Weekday.eSunday;
	
	tEntry1Time		: TIME;
	fEntry1Value	: REAL;
	tEntry2Time		: TIME;
	fEntry2Value	: REAL;
	tEntry3Time		: TIME;
	fEntry3Value	: REAL;
END_VAR

F_BA_SetWeekdays(F_BACnet_SchedWeekly3xA, eDayFrom, eDayTo, 1, tEntry1Time, F_BA_RVal(fEntry1Value));
F_BA_SetWeekdays(F_BACnet_SchedWeekly3xA, eDayFrom, eDayTo, 2, tEntry2Time, F_BA_RVal(fEntry2Value));
F_BA_SetWeekdays(F_BACnet_SchedWeekly3xA, eDayFrom, eDayTo, 3, tEntry3Time, F_BA_RVal(fEntry3Value));

END_FUNCTION

// POUs/Helper/Scheduler/Weekly/F_BACnet_SchedWeekly3xB
// Returns an initialized binary weekly scheduler.
FUNCTION F_BACnet_SchedWeekly3xB : T_BACnet_SchedWeek
VAR_INPUT
	eDayFrom		: E_BA_Weekday		:= E_BA_Weekday.eMonday;
	eDayTo			: E_BA_Weekday		:= E_BA_Weekday.eSunday;
	
	tEntry1Time		: TIME;
	bEntry1Value	: BOOL;
	tEntry2Time		: TIME;
	bEntry2Value	: BOOL;
	tEntry3Time		: TIME;
	bEntry3Value	: BOOL;
END_VAR

F_BA_SetWeekdays(F_BACnet_SchedWeekly3xB, eDayFrom, eDayTo, 1, tEntry1Time, F_BA_BVal(bEntry1Value));
F_BA_SetWeekdays(F_BACnet_SchedWeekly3xB, eDayFrom, eDayTo, 2, tEntry2Time, F_BA_BVal(bEntry2Value));
F_BA_SetWeekdays(F_BACnet_SchedWeekly3xB, eDayFrom, eDayTo, 3, tEntry3Time, F_BA_BVal(bEntry3Value));

END_FUNCTION

// POUs/Helper/Scheduler/Weekly/F_BACnet_SchedWeekly3xM
// Returns an initialized multistate weekly scheduler.
FUNCTION F_BACnet_SchedWeekly3xM : T_BACnet_SchedWeek
VAR_INPUT
	eDayFrom		: E_BA_Weekday		:= E_BA_Weekday.eMonday;
	eDayTo			: E_BA_Weekday		:= E_BA_Weekday.eSunday;
	
	tEntry1Time		: TIME;
	nEntry1Value	: UDINT;
	tEntry2Time		: TIME;
	nEntry2Value	: UDINT;
	tEntry3Time		: TIME;
	nEntry3Value	: UDINT;
END_VAR

F_BA_SetWeekdays(F_BACnet_SchedWeekly3xM, eDayFrom, eDayTo, 1, tEntry1Time, F_BA_UDIVal(nEntry1Value));
F_BA_SetWeekdays(F_BACnet_SchedWeekly3xM, eDayFrom, eDayTo, 2, tEntry2Time, F_BA_UDIVal(nEntry2Value));
F_BA_SetWeekdays(F_BACnet_SchedWeekly3xM, eDayFrom, eDayTo, 3, tEntry3Time, F_BA_UDIVal(nEntry3Value));

END_FUNCTION

// POUs/Helper/Scheduler/Weekly/F_BACnet_SchedWeekly5xA
// Returns an initialized analog weekly scheduler.
FUNCTION F_BACnet_SchedWeekly5xA : T_BACnet_SchedWeek
VAR_INPUT
	eDayFrom		: E_BA_Weekday		:= E_BA_Weekday.eMonday;
	eDayTo			: E_BA_Weekday		:= E_BA_Weekday.eSunday;
	
	tEntry1Time		: TIME;
	fEntry1Value	: REAL;
	tEntry2Time		: TIME;
	fEntry2Value	: REAL;
	tEntry3Time		: TIME;
	fEntry3Value	: REAL;
	tEntry4Time		: TIME;
	fEntry4Value	: REAL;
	tEntry5Time		: TIME;
	fEntry5Value	: REAL;
END_VAR

F_BA_SetWeekdays(F_BACnet_SchedWeekly5xA, eDayFrom, eDayTo, 1, tEntry1Time, F_BA_RVal(fEntry1Value));
F_BA_SetWeekdays(F_BACnet_SchedWeekly5xA, eDayFrom, eDayTo, 2, tEntry2Time, F_BA_RVal(fEntry2Value));
F_BA_SetWeekdays(F_BACnet_SchedWeekly5xA, eDayFrom, eDayTo, 3, tEntry3Time, F_BA_RVal(fEntry3Value));
F_BA_SetWeekdays(F_BACnet_SchedWeekly5xA, eDayFrom, eDayTo, 4, tEntry4Time, F_BA_RVal(fEntry4Value));
F_BA_SetWeekdays(F_BACnet_SchedWeekly5xA, eDayFrom, eDayTo, 5, tEntry5Time, F_BA_RVal(fEntry5Value));

END_FUNCTION

// POUs/Helper/Scheduler/Weekly/F_BACnet_SchedWeekly5xB
// Returns an initialized binary weekly scheduler.
FUNCTION F_BACnet_SchedWeekly5xB : T_BACnet_SchedWeek
VAR_INPUT
	eDayFrom		: E_BA_Weekday		:= E_BA_Weekday.eMonday;
	eDayTo			: E_BA_Weekday		:= E_BA_Weekday.eSunday;
	
	tEntry1Time		: TIME;
	bEntry1Value	: BOOL;
	tEntry2Time		: TIME;
	bEntry2Value	: BOOL;
	tEntry3Time		: TIME;
	bEntry3Value	: BOOL;
	tEntry4Time		: TIME;
	bEntry4Value	: BOOL;
	tEntry5Time		: TIME;
	bEntry5Value	: BOOL;
END_VAR

F_BA_SetWeekdays(F_BACnet_SchedWeekly5xB, eDayFrom, eDayTo, 1, tEntry1Time, F_BA_BVal(bEntry1Value));
F_BA_SetWeekdays(F_BACnet_SchedWeekly5xB, eDayFrom, eDayTo, 2, tEntry2Time, F_BA_BVal(bEntry2Value));
F_BA_SetWeekdays(F_BACnet_SchedWeekly5xB, eDayFrom, eDayTo, 3, tEntry3Time, F_BA_BVal(bEntry3Value));
F_BA_SetWeekdays(F_BACnet_SchedWeekly5xB, eDayFrom, eDayTo, 4, tEntry4Time, F_BA_BVal(bEntry4Value));
F_BA_SetWeekdays(F_BACnet_SchedWeekly5xB, eDayFrom, eDayTo, 5, tEntry5Time, F_BA_BVal(bEntry5Value));

END_FUNCTION

// POUs/Helper/Scheduler/Weekly/F_BACnet_SchedWeekly5xM
// Returns an initialized multistate weekly scheduler.
FUNCTION F_BACnet_SchedWeekly5xM : T_BACnet_SchedWeek
VAR_INPUT
	eDayFrom		: E_BA_Weekday		:= E_BA_Weekday.eMonday;
	eDayTo			: E_BA_Weekday		:= E_BA_Weekday.eSunday;
	
	tEntry1Time		: TIME;
	nEntry1Value	: UDINT;
	tEntry2Time		: TIME;
	nEntry2Value	: UDINT;
	tEntry3Time		: TIME;
	nEntry3Value	: UDINT;
	tEntry4Time		: TIME;
	nEntry4Value	: UDINT;
	tEntry5Time		: TIME;
	nEntry5Value	: UDINT;
END_VAR

F_BA_SetWeekdays(F_BACnet_SchedWeekly5xM, eDayFrom, eDayTo, 1, tEntry1Time, F_BA_UDIVal(nEntry1Value));
F_BA_SetWeekdays(F_BACnet_SchedWeekly5xM, eDayFrom, eDayTo, 2, tEntry2Time, F_BA_UDIVal(nEntry2Value));
F_BA_SetWeekdays(F_BACnet_SchedWeekly5xM, eDayFrom, eDayTo, 3, tEntry3Time, F_BA_UDIVal(nEntry3Value));
F_BA_SetWeekdays(F_BACnet_SchedWeekly5xM, eDayFrom, eDayTo, 4, tEntry4Time, F_BA_UDIVal(nEntry4Value));
F_BA_SetWeekdays(F_BACnet_SchedWeekly5xM, eDayFrom, eDayTo, 5, tEntry5Time, F_BA_UDIVal(nEntry5Value));

END_FUNCTION

// POUs/Helper/String/F_BACnet_GetObjectIdString
FUNCTION F_BACnet_GetObjectIdString : STRING
VAR_INPUT
	tObjectID : T_BACnet_ObjectIdentifier := 16#FFFFFFFF;
END_VAR
VAR
	nObjType	: DINT;
	nObjInstance: UDINT;
END_VAR

nObjType	:= F_BACnet_GetObjType(tObjectID);
nObjInstance:= F_BACnet_GetObjInstance(tObjectID);
IF (BACnet_Globals.nRange_ObjectTypeFirst <= nObjType) AND (nObjType <= BACnet_Globals.nRange_ObjectTypeLast) THEN
	F_BACnet_GetObjectIdString := CONCAT(CONCAT(BACnet_Globals.sSpec_ObjectTypeShortcut[nObjType], ':'), UDINT_TO_STRING(nObjInstance));
ELSE
	F_BACnet_GetObjectIdString := CONCAT('???:', UDINT_TO_STRING(nObjInstance));
END_IF

END_FUNCTION

// POUs/Helper/F_BACnet_GetObjType
FUNCTION F_BACnet_GetObjType : E_BACnetObjType
VAR_INPUT
	nObjectId : DWORD;
END_VAR
VAR
END_VAR

F_BACnet_GetObjType := TO_INT(SHR((nObjectId AND 16#FFC00000), 22));

END_FUNCTION

// POUs/Helper/String/FB_BACnet_StringExtDecode
FUNCTION_BLOCK FB_BACnet_StringExtDecode (* convert UTF-8/UCS2/UCS4/ISO8859-1 to Windows-1252 *)
VAR_INPUT
	pChrStringExt	: POINTER TO ST_BACnet_CharacterStringExt; (* BACnet character string data structure (header and string) *)
	pOutString		: POINTER TO T_MaxString; (* pointer to result buffer (Windows-1252 encoded) *)
	nOutSize		: UDINT; (* byte size *)
END_VAR
VAR_OUTPUT
	bValid			: BOOL; (* Decoding successfull *)
	bOverflow		: BOOL; (* String length overflow (source string too long) *)
	bUnsupported	: BOOL; (* Souce encoding is unsupported (use ReadProp function and decode manually instead) *)
	nLength			: UDINT; (* out character length *)
	eSrcEncoding	: E_BACnet_StringEncodingTypes; (* input encoding *)
END_VAR
VAR
	pText 			: POINTER TO BYTE;
	pByte			: POINTER TO BYTE;
END_VAR

(* preset valid to FALSE *)
bValid := FALSE;
bOverflow := FALSE;
bUnsupported := FALSE;
(* check pointer *)
IF (pChrStringExt = 0) OR (pOutString = 0) THEN
	nLength := 0;
(* check input size *)
ELSIF (nOutSize = 0) THEN
	(* NULL string *)
	bValid := TRUE;
	pOutString^ := '';
	nLength := 0;
	eSrcEncoding := E_BACnet_StringEncodingTypes.eAnsiUtf8;
ELSE
	(* string data available *)
	IF (pChrStringExt^.cookie = 0) THEN
		(* new character string type *)
		nLength			:= UDINT_TO_UINT(pChrStringExt^.strLen);
		eSrcEncoding	:= UDINT_TO_INT(pChrStringExt^.encoding);
		pText			:= ADR(pChrStringExt^.stringData);
	ELSE
		(* ASCII/UTF-8 string *)
		nLength			:= F_BACnet_ChrStrExtLen(pChrStringExt^);
		eSrcEncoding	:= E_BACnet_StringEncodingTypes.eAnsiUtf8;
		pText			:= pChrStringExt;
	END_IF

	(* check size *)
	IF (nLength = 0) THEN
		(* no data *)
		bValid := TRUE;
		pOutString^ := '';
	ELSIF (nLength <= nOutSize) THEN
		(* copy to output buffer first *)
		MEMMOVE(destAddr:= pOutString, srcAddr:= pText, n:= nLength);

		(* decode and copy *)
		CASE eSrcEncoding OF

			E_BACnet_StringEncodingTypes.eAnsiUtf8:
				bValid := TRUE;
				nLength := UDINT_TO_UINT(F_BACnet_DecodeUTF8(pOutString, nLength));

			E_BACnet_StringEncodingTypes.eUCS2:
				bValid := TRUE;
				nLength := UDINT_TO_UINT(F_BACnet_DecodeUCS2(pOutString, nLength));

			E_BACnet_StringEncodingTypes.eUCS4:
				bValid := TRUE;
				nLength := UDINT_TO_UINT(F_BACnet_DecodeUCS4(pOutString, nLength));

			E_BACnet_StringEncodingTypes.eISO8859:
				bValid := TRUE;
				(* check if string termination is already part of string *)
				pByte := pOutString + nLength - 1;
				IF (pByte^ = 16#00) THEN
					(* termination already part of string *)
					nLength := nLength - 1;
				ELSE
					(* add string termination *)
					pByte := pOutString + nLength;
					pByte^ := 16#00;
				END_IF

			ELSE
				bUnsupported := TRUE;

		END_CASE
	ELSE
		(* text too long *)
		nLength := 0;
		pOutString^ := '';
		bOverflow := TRUE;
	END_IF
END_IF

END_FUNCTION_BLOCK

// POUs/Helper/String/FB_BACnet_StringExtEncode
FUNCTION_BLOCK FB_BACnet_StringExtEncode (* convert Windows-1252 to ANSI/UTF-8 BACnet Character String *)
VAR_INPUT
	pString			: POINTER TO T_MaxString; (* pointer to Windows-1252 encoded PLC text *)
	nSize			: INT; (* string length or data size of pText field *)
	pResultExtStr	: POINTER TO ST_BACnet_CharacterStringExt;
	nResult		: UDINT; (* byte size of result data field *)
END_VAR
VAR_OUTPUT
	bValid			: BOOL;
	bOverflow		: BOOL; (* String length overflow (source string too long) *)
	nLength			: UDINT; (* out string data length in byte *)
END_VAR

(* preset valid to FALSE *)
bOverflow := FALSE;
bValid := TRUE;
(* check pointer *)
IF (pString = 0) OR (pResultExtStr = 0) THEN
	nLength := 0;
	bValid := FALSE;
	RETURN;
END_IF

(* clear string *)
MEMSET(destAddr:=pResultExtStr, fillByte:=0, n:=nResult);
(* check input size *)
IF (nSize <= 0) THEN
	nLength := 0;

(* convert *)
ELSE
	IF (F_BACnet_EncodeUTF8(
		pString		:= pString,
		nString	:= TO_UDINT(nSize),
		pResult		:= pResultExtStr,
		nResult	:= nResult,
		nResultLen	:= nLength) > nResult)
	THEN
		bOverflow	:= TRUE;
		bValid		:= FALSE;
	END_IF
END_IF

END_FUNCTION_BLOCK

// POUs/Helper/F_BACnet_GetObjectListIndex
FUNCTION F_BACnet_GetObjectListIndex : DINT
VAR_INPUT
	tObjectId	: T_BACnet_ObjectIdentifier := 16#FFFFFFFF;
END_VAR

VAR
	nMax : DINT;
	i : DINT;
END_VAR
(*All VAR_IN_OUT variables have been moved to the end of the declaration due to compatibility reasons*)
VAR_IN_OUT
	stObjIDList	: ST_BACnet_ObjectIdentifierList;
END_VAR

nMax := UDINT_TO_DINT(stObjIDList.nEntries)-1;
F_BACnet_GetObjectListIndex := -1; (* preset: no match *)
FOR i := 0 TO nMax DO
	IF stObjIDList.arrObjList[i] = tObjectId THEN
		F_BACnet_GetObjectListIndex := i; (* match *)
		RETURN;
	END_IF
END_FOR

END_FUNCTION

// POUs/Helper/FB_BACnet_AccLimit
FUNCTION_BLOCK FB_BACnet_AccLimit
VAR_INPUT
	X : REAL; (* input value [1] *)
	Amax : REAL; (* maximum acceleration of X [1/s]; 0 = limit disabled *)
	Tcycle : REAL; (* cycle time [s] of task; 0 = use internal measuring *)
END_VAR
VAR_OUTPUT
	Y : REAL; (* limited X value [1] *)
	A : REAL; (* input acceleration [1/s] *)
END_VAR
VAR
	_sysTime	: GETCPUCOUNTER;
	_Time		: T_LARGE_INTEGER;
	_TimeOld	: T_LARGE_INTEGER;
	_tCycleTime	: REAL;
	_bFirstScan	: BOOL:=TRUE;
	_foldY		: REAL;
END_VAR

(* determine cycle time *)
IF Tcycle = 0.0 THEN
	_TimeOld := _Time;
	_sysTime(cpuCntLoDW=> _Time.dwLowPart, cpuCntHiDW=> _Time.dwHighPart);
	_tCycleTime := F_BACnet_SysTimeDiff(In1:=_Time, In2:=_TimeOld);
ELSE
	_tCycleTime := Tcycle;
END_IF

IF (NOT _bFirstScan) THEN
	(* exit on wrong cycle time *)
	IF _tCycleTime <= 0.0 THEN
		RETURN;
	END_IF
	(* calculate current acceleration *)
	A := (X - _foldY) / _tCycleTime;
	IF (Amax <> 0.0) THEN
		Amax := ABS(Amax);
		IF (ABS(A) > Amax) THEN
			IF (A >= 0.0) THEN
				Y := _foldY + (Amax * _tCycleTime);
			ELSE
				Y := _foldY - (Amax * _tCycleTime);
			END_IF
		ELSE
			Y := X;
		END_IF
	ELSE
		Y := X;
	END_IF
ELSE
	Y := X;
END_IF

_foldY := Y;
_bFirstScan:=FALSE;

END_FUNCTION_BLOCK

// POUs/Helper/FB_BACnet_AvgValue
FUNCTION_BLOCK FB_BACnet_AvgValue
VAR_INPUT
	X	: REAL; (* input value to average *)
	n	: UINT; (* number of averages (0 = no average --> Y = X) *)
END_VAR
VAR_OUTPUT
	Y	: REAL; (* average result *)
END_VAR
VAR
	_n	: UINT := 0;
	_Xn : LREAL;
END_VAR

IF (_n > n) THEN
	_n := n;
END_IF
IF (_n = 0) OR (n = 0) THEN
	_Xn := REAL_TO_LREAL(X);
ELSE
	_Xn := ((_Xn * _n) + REAL_TO_LREAL(X)) / UINT_TO_LREAL(_n + 1);
END_IF
_n := _n + 1;
Y := LREAL_TO_REAL(_Xn);

END_FUNCTION_BLOCK

// POUs/Helper/FB_BACnet_PidControl
FUNCTION_BLOCK FB_BACnet_PidControl
VAR_INPUT
	(* controller input  *)
	fSetpoint				: REAL;	(* setpoint value *)
	fPresentValue			: REAL;	(* actual value *)
	(* reset flag *)
	bReset					: BOOL;
	(* controller values *)
	fCtrlCycleTime			: REAL; (* controller cycle time in seconds [s] *)

	fBias					: REAL; (* bias also active when reset is set to 1 *)
	fKp						: REAL;	(* proportional gain Kp	(P) *)
	fKi						: REAL; (* integral gain Ki (I) *)
	fKd						: REAL;	(* derivative gain Kd (D) *)
	fTp						: REAL := -1.0;	(* damping time Tp (PT1) [s] (fTp < 0 --> Tp = Kd / 10) *)

	(* maximum ratings *)
	fMaxOutput				: REAL;
	fMinOutput				: REAL;
END_VAR
VAR_OUTPUT
	fY						: REAL; (* controller output command *)
	eErrorStatus			: E_BACnet_Error;
END_VAR
VAR
	(* Internal Variable *)
	_fE		: REAL;
	_fEOld	: REAL;
	_fYp	: REAL;
	_fYi	: REAL;
	_fYd	: REAL;
	_fbYd	: FB_BACnet_PT1;
END_VAR

(* preset error number *)
eErrorStatus	:= E_BACnet_Error.eNoError;

(* check cycle time parameter: (CycleTime > 0) *)
IF (fCtrlCycleTime <= 0.0) THEN
	eErrorStatus := E_BACnet_Error.eInvalidCycleTime;
	bReset := TRUE;
END_IF;

(* check controller parameters: (Kp, Ki, Kd >= 0) *)
IF ((fKp < 0.0) OR (fKi < 0.0) OR (fKd < 0.0)) THEN
	eErrorStatus := E_BACnet_Error.eInvalidParameter;
	bReset := TRUE;
END_IF;

(* controller reset *)
IF bReset THEN
	(* reset internal and external variables *)
	_fEOld	:= 0.0;
	fY		:= MAX(MIN(fBias, fMaxOutput), fMinOutput);
	_fYi	:= 0.0;
	_fbYd(X:= 0.0, T:= 0.0, Y=> );
	RETURN;
END_IF

(* 3. save old variable *)
_fEOld := _fE;

(* 4. set error/deviation input *)
_fE := fSetpoint - fPresentValue;

(* 5. YP-part *)
_fYp := fKp * _fE;

(* 6. YI-part *)
IF (fKi = 0.0) THEN
	_fYi	:= 0.0;
ELSE
	_fYi := _fYi + (fKi * fCtrlCycleTime * _fE);
END_IF
IF (_fYi > fMaxOutput) THEN
	(* limit wind up positive *)
	_fYi := fMaxOutput;
ELSIF (_fYi < fMinOutput) THEN
	(* limit wind up negative *)
	_fYi := fMinOutput;
END_IF

(* 7. YD-part *)
IF (fTp < 0.0) THEN
	fTp := fKd / 10.0;
END_IF
_fYd := fKd * (_fE - _fEOld) / fCtrlCycleTime;
_fbYd(X:= _fYd, T:= fTp, Tcycle:= fCtrlCycleTime, Y=> );

(* 8. Ysum = YP + YI + YD + Bias and output *)
fY := _fYp + _fYi + _fbYd.Y + fBias;
fY := MAX(MIN(fY, fMaxOutput), fMinOutput);

END_FUNCTION_BLOCK

// POUs/Helper/FB_BACnet_PT1
FUNCTION_BLOCK FB_BACnet_PT1
VAR_INPUT
	X : REAL; (* input value *)
	T : REAL; (* damping time [s] *)
	Tcycle : REAL; (* cycle time [s] of task; 0 = use internal measuring *)
END_VAR
VAR_OUTPUT
	Y : REAL; (* damped value *)
END_VAR
VAR
	_sysTime	: GETCPUCOUNTER;
	_Time		: T_LARGE_INTEGER;
	_TimeOld	: T_LARGE_INTEGER;
	_tCycleTime	: REAL;
	_Yold : REAL;
	_FirstScan : BOOL := TRUE;
END_VAR

(* determine cycle time *)
IF Tcycle = 0.0 THEN
	_TimeOld := _Time;
	_sysTime(cpuCntLoDW=> _Time.dwLowPart, cpuCntHiDW=> _Time.dwHighPart);
	_tCycleTime := F_BACnet_SysTimeDiff(In1:=_Time, In2:=_TimeOld);
ELSE
	_tCycleTime := Tcycle;
END_IF

(* exit on wrong cycle time *)
IF _tCycleTime <= 0.0 THEN
	RETURN;
END_IF

(* initialize and check on zero/negative damping time *)
IF (T <= 0.0) OR _FirstScan THEN
	Y := X;
	_Yold := Y;
	_FirstScan := FALSE;
	RETURN;
END_IF

(* remind last result *)
_Yold := Y;

(* calculate result *)
Y := 1 / ((T / _tCycleTime) + 1) * (X - _Yold) + _Yold;

END_FUNCTION_BLOCK

// POUs/Local/Objects/[Base]/Basic/FB_BACnet_EventObject
FUNCTION_BLOCK FB_BACnet_EventObject EXTENDS FB_BACnet_Object
VAR_INPUT CONSTANT PERSISTENT
	{region 'Variable Parameters'}
		{attribute 'parameterCategory':='EventConfig'}
		bEventDetectionEnable : BOOL := TRUE;
		
		{attribute 'parameterCategory':='EventConfig'}
		nNotificationClass : UDINT;
		{attribute 'parameterCategory':='EventConfig'}
		eNotifyType : E_BACnet_NotifyType := E_BACnet_NotifyType.eAlarm;
		{attribute 'parameterCategory':='EventConfig'}
		bEventEnable : ARRAY[E_BA_EventTransition.First .. E_BA_EventTransition.Last] OF BOOL;
		{attribute 'parameterCategory':='EventConfig'}
		sEventMessageTextsConfig : ARRAY[E_BA_EventTransition.First .. E_BA_EventTransition.Last] OF T_MaxString;
		{attribute 'parameterCategory':='EventConfig'}
		nTimeDelay : UDINT;
		{attribute 'parameterCategory':='EventConfig'}
		nTimeDelayNormal : UDINT;
	{endregion}
END_VAR
VAR_INPUT CONSTANT
	{region 'Operational Parameters'}
		{attribute 'parameterCategory':='Event'}
		bAcknowledgeRm : BOOL;														// Acknowledge outstanding event transition states (from remote via parameter).
	{endregion}
END_VAR
VAR_OUTPUT
	bEvent						: BOOL;												// Indicates an active event
	eReliability				: E_BACnet_Reliability;
END_VAR
VAR
	{region 'Event'}
		stStateFlags			: ST_BA_StatusFlags;
		stAckedTransitions		: ST_BA_EventTransitions;

		eEventState				: E_BACnet_EventState;
	{endregion}
	{region 'Misc'}
		rAckPLCTrig				: R_TRIG;
	{endregion}
END_VAR

rAckPLCTrig();
IF (rAckPLCTrig.Q) THEN
	// Acknowledge all event states:
	Acknowledge(E_BA_EventTransition.Invalid, BACnet_Param.sEvtMgmt_AckMsgPLC);
END_IF
IF bAcknowledgeRm THEN
	bAcknowledgeRm := FALSE;
	// Acknowledge all event states:
	Acknowledge(E_BA_EventTransition.Invalid, BACnet_Param.sEvtMgmt_AckMsgRemote);
END_IF

SUPER^();

bEvent := F_BA_IsDisturbed(stStateFlags);

METHOD PROTECTED OnObjectStateChanged
SUPER^.OnObjectStateChanged();

CASE (tState) OF
	TCOM_STATE.TCOM_STATE_PREOP:
		// SyncHandler:
		RequestSyncHandlers(9, 11);
		
		// Properties:
		EnableProperty(E_BACnetPropIdentifier.PropEventAlgorithmInhibit, FALSE);
		EnableProperty(E_BACnetPropIdentifier.PropReliabilityEvaluationInhibit, FALSE);
		
		// Ensure UTF-8 Encoding:
		F_BA_EnsureUTF8Array(ADR(sEventMessageTextsConfig), SIZEOF(sEventMessageTextsConfig[1]), TO_DINT(E_BA_EventTransition.Count));
		
	TCOM_STATE.TCOM_STATE_SAFEOP:
		;
	
	TCOM_STATE.TCOM_STATE_OP:
		ConcatTitle(sEventMessageTextsConfig[E_BA_EventTransition.eToOffnormal], sDescription, BACnet_Param.sSeparator_EventMessageText);
		ConcatTitle(sEventMessageTextsConfig[E_BA_EventTransition.eToFault], sDescription, BACnet_Param.sSeparator_EventMessageText);
		ConcatTitle(sEventMessageTextsConfig[E_BA_EventTransition.eToNormal], sDescription, BACnet_Param.sSeparator_EventMessageText);
		
		// Synchronize:
		SyncProperty(E_BACnetPropIdentifier.PropEventDetectionEnable, SIZEOF(bEventDetectionEnable), ADR(bEventDetectionEnable), 0, eFullSync_InitPLC, FALSE);
		SyncProperty(E_BACnetPropIdentifier.PropNotificationClass, SIZEOF(nNotificationClass), ADR(nNotificationClass), 0, eFullSync_InitPLC, FALSE);
		SyncProperty(E_BACnetPropIdentifier.PropNotifyType, SIZEOF(eNotifyType), ADR(eNotifyType), 0, eFullSync_InitPLC, FALSE);
		SyncPropertyIdx(E_BACnetPropIdentifier.PropEventEnable, SIZEOF(BOOL), ADR(bEventEnable[E_BA_EventTransition.eToOffnormal]), E_BACnet_EventTransitionBits.eToOffnormal, 0, eFullSync_InitPLC, FALSE);	
		SyncPropertyIdx(E_BACnetPropIdentifier.PropEventEnable, SIZEOF(BOOL), ADR(bEventEnable[E_BA_EventTransition.eToFault]), E_BACnet_EventTransitionBits.eToFault, 0, eFullSync_InitPLC, FALSE);	
		SyncPropertyIdx(E_BACnetPropIdentifier.PropEventEnable, SIZEOF(BOOL), ADR(bEventEnable[E_BA_EventTransition.eToNormal]), E_BACnet_EventTransitionBits.eToNormal, 0, eFullSync_InitPLC, FALSE);
		SyncPropertyIdx(E_BACnetPropIdentifier.PropEventMessageTextsConfig, SIZEOF(T_MaxString), ADR(sEventMessageTextsConfig[E_BA_EventTransition.eToOffnormal]), (E_BACnet_EventTransitionBits.eToOffnormal+1), 0, eFullSync_InitPLC, FALSE);
		SyncPropertyIdx(E_BACnetPropIdentifier.PropEventMessageTextsConfig, SIZEOF(T_MaxString), ADR(sEventMessageTextsConfig[E_BA_EventTransition.eToFault]), (E_BACnet_EventTransitionBits.eToFault+1), 0, eFullSync_InitPLC, FALSE);
		SyncPropertyIdx(E_BACnetPropIdentifier.PropEventMessageTextsConfig, SIZEOF(T_MaxString), ADR(sEventMessageTextsConfig[E_BA_EventTransition.eToNormal]), (E_BACnet_EventTransitionBits.eToNormal+1), 0, eFullSync_InitPLC, FALSE);
		
		IF (eObjectType <> E_BACnetObjType.ObjTrendLog) AND (eObjectType <> E_BACnetObjType.ObjTrendLogMultiple) THEN
			SyncProperty(E_BACnetPropIdentifier.PropTimeDelay, SIZEOF(nTimeDelay), ADR(nTimeDelay), 0, eFullSync_InitPLC, FALSE);
			SyncProperty(E_BACnetPropIdentifier.PropTimeDelayNormal, SIZEOF(nTimeDelayNormal), ADR(nTimeDelayNormal), 0, eFullSync_InitPLC, FALSE);
		END_IF
		
		SyncPropertyIdx(E_BACnetPropIdentifier.PropStatusFlags, SIZEOF(BOOL), ADR(stStateFlags.bOverridden), E_BACnet_StatusFlags.eOverridden, 0, eSync_FromSupplement, FALSE);	
		SyncPropertyIdx(E_BACnetPropIdentifier.PropStatusFlags, SIZEOF(BOOL), ADR(stStateFlags.bOutOfService), E_BACnet_StatusFlags.eOutOfService, 0, eSync_FromSupplement, FALSE);	
		SyncPropertyIdx(E_BACnetPropIdentifier.PropStatusFlags, SIZEOF(BOOL), ADR(stStateFlags.bFault), E_BACnet_StatusFlags.eFault, 0, eSync_FromSupplement, FALSE);	
		SyncPropertyIdx(E_BACnetPropIdentifier.PropStatusFlags, SIZEOF(BOOL), ADR(stStateFlags.bInAlarm), E_BACnet_StatusFlags.eInAlarm, 0, eSync_FromSupplement, FALSE);
		SyncPropertyIdx(E_BACnetPropIdentifier.PropAckedTransitions, SIZEOF(BOOL), ADR(stAckedTransitions.bToOffnormal), E_BACnet_EventTransitionBits.eToOffnormal, 0, eSync_FromSupplement, FALSE);	
		SyncPropertyIdx(E_BACnetPropIdentifier.PropAckedTransitions, SIZEOF(BOOL), ADR(stAckedTransitions.bToFault), E_BACnet_EventTransitionBits.eToFault, 0, eSync_FromSupplement, FALSE);	
		SyncPropertyIdx(E_BACnetPropIdentifier.PropAckedTransitions, SIZEOF(BOOL), ADR(stAckedTransitions.bToNormal), E_BACnet_EventTransitionBits.eToNormal, 0, eSync_FromSupplement, FALSE);	
		SyncProperty(E_BACnetPropIdentifier.PropReliability, SIZEOF(eReliability), ADR(eReliability), 0, eSync_FromSupplement, FALSE);
		SyncProperty(E_BACnetPropIdentifier.PropEventState, SIZEOF(eEventState), ADR(eEventState), 0,  eSync_FromSupplement, FALSE);
		
END_CASE
END_METHOD

METHOD FB_init : BOOL
VAR_INPUT
	bInitRetains : BOOL; // if TRUE, the retain variables are initialized (warm start / cold start)
	bInCopyCode : BOOL;  // if TRUE, the instance afterwards gets moved into the copy code (online change)
END_VAR
IF (bInitRetains) THEN
	// Indicate inheritance of event message texts as default:
	sEventMessageTextsConfig[E_BA_EventTransition.eToOffnormal] := CONCAT(BACnet_Globals.sCmd_ConcatTitle, 'To Off-Normal');
	sEventMessageTextsConfig[E_BA_EventTransition.eToFault] := CONCAT(BACnet_Globals.sCmd_ConcatTitle, 'To Fault');
	sEventMessageTextsConfig[E_BA_EventTransition.eToNormal] := CONCAT(BACnet_Globals.sCmd_ConcatTitle, 'To Normal');
END_IF
END_METHOD

// Acknowledge via Property.
// > This property is triggered (Only rising edges acknowledges current instance!)
PROPERTY AcknowledgePLC : BOOL
GET
AcknowledgePLC := rAckPLCTrig.CLK;
END_GET
SET
rAckPLCTrig.CLK := AcknowledgePLC;
END_SET
END_PROPERTY

PROPERTY AcknowledgeRm : BOOL
GET
AcknowledgeRm := bAcknowledgeRm;
END_GET
SET
bAcknowledgeRm := AcknowledgeRm;
END_SET
END_PROPERTY

PROPERTY IsReliable : BOOL
GET
IsReliable := (eReliability = E_BACnet_Reliability.eNoFaultDetected) AND (NOT stStateFlags.bOverridden) AND (NOT stStateFlags.bOutOfService);
END_GET
END_PROPERTY

PROPERTY AckedTransitions : ST_BA_EventTransitions
GET
AckedTransitions := stAckedTransitions;
END_GET
END_PROPERTY

PROPERTY EventState : E_BACnet_EventState
GET
EventState := eEventState;
END_GET
END_PROPERTY

PROPERTY StateFlags : ST_BA_StatusFlags
GET
StateFlags := stStateFlags;
END_GET
END_PROPERTY

END_FUNCTION_BLOCK

// POUs/Local/Objects/[Base]/Basic/FB_BACnet_Object
{attribute 'reflection'}
FUNCTION_BLOCK FB_BACnet_Object EXTENDS FB_BACnet_BaseObject IMPLEMENTS I_BACnet_Object, I_BACnet_ObjectOwner
VAR_INPUT CONSTANT PERSISTENT
	{region 'Variable Parameters'}
		{attribute 'parameterCategory':='General'}
		{attribute 'TcEncoding':='UTF-8'}
		sObjectName : T_MaxString;
		{attribute 'parameterCategory':='General'}
		{attribute 'TcEncoding':='UTF-8'}
		sDescription : T_MaxString;
	{endregion}
END_VAR
VAR
	{region 'UserInit'}
		iParent						: I_BACnet_View;
	{endregion}
END_VAR
VAR
	{region 'COV'}
		bObjNameChanged				: BOOL;
		bDescriptionChanged			: BOOL;
	{endregion}
	{region 'General'}
		{attribute 'instance-path'}
		{attribute 'no_init'}
		sSymbolPath  				: T_MaxString;														// Full symbol path of current instance
		sSymbolName  				: STRING;															// Symbol name of current instance
	{endregion}
	{region 'Internal'}
		{attribute 'hide'}
		bParentInit					: BOOL := TRUE;
		{attribute 'hide'}
		fbLogMsg					: FB_BA_LogMessage;
	{endregion}
END_VAR
VAR CONSTANT
	{region 'Payload-Balancing'}
		{attribute 'hide'}
		COV_UPDATE_CYCLE			: UDINT	:= 100;														// Execute COV-indication every X cycles to ALL properties
		{attribute 'hide'}
		COV_UPDATE_SPLIT			: UDINT	:= 100;														// Splits all objects in max. X groups to execute COV-indication
	{endregion}
END_VAR

IF bReady THEN
	// Request COV-Update:
	bUpdateCOV := (nUpdateCount MOD COV_UPDATE_CYCLE) = (nObjectInstance MOD COV_UPDATE_SPLIT);
	
	SUPER^();
	
	IF bParentInit THEN
		IF iParent = 0 THEN
			bParentInit := FALSE;
		ELSE
			// Wait for parent to get initialized:
			IF iParent.Ready THEN
				__QUERYPOINTER(iParent, _fbViewTmp);
				_fbViewTmp^.View_RegisterChildObject(THIS^);
		
				bParentInit := FALSE;
			END_IF
		END_IF
	ELSE
		// Concatenate changed titles at runtime:
		ValidateTitles();
	END_IF
ELSE
	SUPER^();
END_IF

// Unused - Implemented for compatibility reason!
{attribute 'hide'}
METHOD OnBACnetObjectStateChanged
VAR_INPUT
	tState			: TCOM_STATE;
END_VAR
END_METHOD

METHOD PROTECTED OnObjectStateChanged
SUPER^.OnObjectStateChanged();

CASE (tState) OF
	TCOM_STATE.TCOM_STATE_PREOP:
		// Ensure UTF-8 Encoding:
		F_BA_EnsureUTF8(ADR(sObjectName), SIZEOF(sObjectName));
		F_BA_EnsureUTF8(ADR(sDescription), SIZEOF(sDescription));
	
		// SyncHandler:
		RequestSyncHandlers(1, 3);

	TCOM_STATE.TCOM_STATE_SAFEOP:
		// Register current instance in server:
		IF (NOT Server.RegisterObject(tObjectID, THIS^)) THEN
			fbLogMsg.Show(ADSLOG_MSGTYPE_ERROR, 'OOSC12', 'Failed to register curernt instance in object list!', FALSE);	
		END_IF
		
	TCOM_STATE.TCOM_STATE_OP:
		// Build titles:
		bObjNameChanged := TRUE;
		bDescriptionChanged := TRUE;
		
		ValidateTitles();
		
		IF S_OK <> SyncProperty(E_BACnetPropIdentifier.PropObjectName, SIZEOF(sObjectName), ADR(sObjectName), ADR(bObjNameChanged), eFullSync_InitPLC, FALSE) THEN
			// Init object name failed!
			// > Try init symbol path instead:
			_hResult := SyncProperty(E_BACnetPropIdentifier.PropObjectName, SIZEOF(sSymbolPath), ADR(sSymbolPath), 0, eFullSync_InitPLC, FALSE);
			IF _hResult = S_OK THEN
				fbLogMsg.Show2(ADSLOG_MSGTYPE_ERROR, 'OOSC26', 'Duplicate use of object name "%s" by "%s"!', F_STRING(sObjectName), F_STRING(sSymbolPath), FALSE);
				sObjectName := sSymbolPath;
			ELSE
				fbLogMsg.Show2(ADSLOG_MSGTYPE_ERROR, 'OOSC29', 'Failed to initialize object name of "%s" (Error: "0x%x")!', F_STRING(sSymbolPath), F_DINT(_hResult), FALSE);
			END_IF
		END_IF
		
		SyncProperty(E_BACnetPropIdentifier.PropDescription, SIZEOF(sDescription), ADR(sDescription), ADR(bDescriptionChanged), eFullSync_InitPLC, FALSE);
		
END_CASE
END_METHOD

METHOD INTERNAL ValidateReference : BOOL
VAR_IN_OUT
	iReference			: I_BACnet_Object;
	tIdentifier			: T_BACnet_ObjectIdentifier;
END_VAR
VAR_INPUT
	eExpectedType		: E_BACnetObjType				:= 16#FF;
END_VAR
VAR
	_bIdentifierValid	: BOOL;
END_VAR
_bIdentifierValid := F_BACnet_IsObjIdentifierValid(tIdentifier);

IF (NOT Ready) THEN
	// Ignore (may persistent stored) pointers:
	iReference := 0;
END_IF
IF (NOT _bIdentifierValid) AND (iReference = 0) THEN
	// Reference undefined:
	ValidateReference := TRUE;
ELSE
	IF (NOT _bIdentifierValid) AND_THEN (iReference <> 0) THEN
		// Interface-pointer of object exists:
		// > Get Object-Identifier:
		tIdentifier := iReference.ObjectID;
		
	ELSIF (_bIdentifierValid) THEN
		// Object identifier of object exists:
		// > Get Interface-pointer:
		IF (NOT Server.GetObject(tIdentifier, iResult=>iReference)) THEN
			tIdentifier := BACnet_Globals.nBACnetObjId_None;
		END_IF
	END_IF
	
	IF (tIdentifier = BACnet_Globals.nBACnetObjId_None) OR (iReference = 0) THEN
		fbLogMsg.Show1(ADSLOG_MSGTYPE_ERROR, 'VOI15', 'Resolving referred object "%d" failed!', F_DWORD(tIdentifier), TRUE);
		
	ELSIF (eExpectedType <> 16#FF) AND_THEN (iReference.ObjectType <> eExpectedType) THEN
		fbLogMsg.Show1(ADSLOG_MSGTYPE_ERROR, 'VOI20', 'Validation of object "%d" failed: type unexpected!', F_DWORD(tIdentifier), TRUE);
			
	ELSE
		ValidateReference := TRUE;
		RETURN;
	END_IF
	
	tIdentifier := 0;
	iReference := 0;
END_IF
END_METHOD

METHOD PROTECTED ConcatTitle : BOOL
VAR_IN_OUT
	sInstTitle			: T_MaxString;
END_VAR
VAR_INPUT
	sParentTitle		: T_MaxString;
	sSeparator			: STRING;
END_VAR
VAR
	iConcatLen			: INT;
END_VAR
iConcatLen := LEN(BACnet_Globals.sCmd_ConcatTitle);

IF (LEFT(sInstTitle, iConcatLen) = BACnet_Globals.sCmd_ConcatTitle) THEN
	// Remove concatenation-command:
	sInstTitle := DELETE(sInstTitle, iConcatLen, 1);
	
	IF (sParentTitle <> '') THEN
		// Concatenate parent title:
		sInstTitle := CONCAT(sSeparator, sInstTitle);
		sInstTitle := CONCAT(sParentTitle, sInstTitle);
	END_IF
END_IF
END_METHOD

METHOD PROTECTED ValidateTitles
// Concatenate titles at runtime:
IF bObjNameChanged THEN
	bObjNameChanged := FALSE;
	ConcatTitle(sObjectName, SEL((iParent <> 0), '', iParent.ObjectName), BACnet_Param.sSeparator_ObjectName);
END_IF
IF bDescriptionChanged THEN
	bDescriptionChanged := FALSE;
	ConcatTitle(sDescription, SEL((iParent <> 0), '', iParent.Description), BACnet_Param.sSeparator_Description);
END_IF
END_METHOD

METHOD FB_init : BOOL
VAR_INPUT
	bInitRetains : BOOL; // if TRUE, the retain variables are initialized (warm start / cold start)
	bInCopyCode : BOOL;  // if TRUE, the instance afterwards gets moved into the copy code (online change)
END_VAR
iOwner := THIS^;

IF (bInitRetains) THEN
	// Remove "Solution Project" title:
	sSymbolPath := right(sSymbolPath, len(sSymbolPath)-find(sSymbolPath,'.'));
	// Remove "PLC Project" title:
	// sSymbolPath := right(sSymbolPath, len(sSymbolPath)-find(sSymbolPath,'.'));
END_IF
	
sSymbolName := F_BA_StringRight(sSymbolPath, '.');
	
fbLogMsg.Path := sSymbolPath;

// Indicate inheritance of project structure as default:
sObjectName := CONCAT(BACnet_Globals.sCmd_ConcatTitle, sSymbolName);
END_METHOD

{attribute 'suppress_wrn_C0410'}
{attribute 'hide'}
PROPERTY LogMsg : REFERENCE TO FB_BA_LogMessage
GET
LogMsg REF= fbLogMsg;
END_GET
END_PROPERTY

PROPERTY Parent : I_BACnet_View
GET
Parent := iParent;
END_GET
SET
IF (iParent = 0) THEN
	iParent := Parent;
ELSE
	fbLogMsg.Show(ADSLOG_MSGTYPE_ERROR, 'P4', 'Object already assigned to parent!', FALSE);
END_IF
END_SET
END_PROPERTY

{attribute 'hide'}
PROPERTY SymbolPath : REFERENCE TO T_MaxString
GET
SymbolPath REF= sSymbolPath;
END_GET
END_PROPERTY

METHOD ReadPropertyExceptionSched : HRESULT
VAR_IN_OUT
	tCalendar			: T_BACnet_SchedCalendar;
	tException			: T_BACnet_SchedExceptionList;
END_VAR
VAR_INPUT
	eDatatype			: E_BACnet_ValueChoice;
END_VAR
VAR
	_i					: INT;
END_VAR
ReadPropertyExceptionSched := SUPER^.ReadPropertyExceptionSched(tCalendar, tException, eDatatype);

IF (ReadPropertyExceptionSched = S_OK) THEN
	// Validate referred objects:
	FOR _i := 1 TO BACnet_Param.nSched_CalendarCount DO
		ValidateReference(tCalendar[_i].iRefCalendar, tCalendar[_i].tRefCalendarID, E_BACnetObjType.ObjCalendar);
	END_FOR
END_IF
END_METHOD

METHOD ReadPropertyReference : HRESULT
VAR_INPUT
	eProperty				: E_BACnetPropIdentifier;
END_VAR
VAR_IN_OUT
	stRefObject				: ST_BACnet_ObjectPropertyReference;
END_VAR
VAR
	stTemp					: ST_BACnet_DeviceObjectPropertyReference;
END_VAR
ReadPropertyReference := SUPER^.ReadPropertyReference(eProperty, stRefObject);

IF (ReadPropertyReference = S_OK) THEN
	ValidateReference(stRefObject.iObject, stRefObject.tObjectID, 16#FF);
END_IF
END_METHOD

METHOD WritePropertyExceptionSched : HRESULT
VAR_IN_OUT
	tCalendar			: T_BACnet_SchedCalendar;
	tException			: T_BACnet_SchedExceptionList;
END_VAR
VAR_INPUT
	eDatatype			: E_BACnet_ValueChoice;
END_VAR
VAR
	_i					: INT;
END_VAR
// Validate referred objects:
FOR _i := 1 TO BACnet_Param.nSched_CalendarCount DO
	ValidateReference(tCalendar[_i].iRefCalendar, tCalendar[_i].tRefCalendarID, E_BACnetObjType.ObjCalendar);
END_FOR

WritePropertyExceptionSched := SUPER^.WritePropertyExceptionSched(tCalendar, tException, eDatatype);
END_METHOD

METHOD WritePropertyReference : HRESULT
VAR_INPUT
	eProperty				: E_BACnetPropIdentifier;
END_VAR
VAR_IN_OUT
	stRefObject				: ST_BACnet_ObjectPropertyReference;
END_VAR
VAR
	stTemp					: ST_BACnet_DeviceObjectPropertyReference;
END_VAR
ValidateReference(stRefObject.iObject, stRefObject.tObjectID, 16#FF);

WritePropertyReference := SUPER^.WritePropertyReference(eProperty, stRefObject);
END_METHOD

PROPERTY Description : T_MaxString
GET
Description := sDescription;
END_GET
SET
sDescription := Description;
END_SET
END_PROPERTY

PROPERTY ObjectName : T_MaxString
GET
ObjectName := sObjectName;
END_GET
SET
sObjectName := ObjectName;
END_SET
END_PROPERTY

END_FUNCTION_BLOCK

// POUs/Local/Objects/[Internal]/FB_BACnet_BaseObject
{attribute 'no_assign'}
{attribute 'hide'}
FUNCTION_BLOCK FB_BACnet_BaseObject IMPLEMENTS I_BACnet_BaseObject
VAR_INPUT CONSTANT
	{region 'Fixed Parameters'}
		{attribute 'parameterCategory':='General'}
		{attribute 'no_copy'}
		Server : REFERENCE TO FB_BACnet_Server := BACnet_Globals.DefaultServer;
		{attribute 'parameterCategory':='General'}
		nObjectInstance : UDINT := 16#003FFFFF;
	{endregion}
END_VAR
VAR
	{region 'Output-Properties'}
		bReady						: BOOL;
	{endregion}
	{region 'SubInit'}
		eObjectType					: E_BACnetObjType				:= 16#FFFF;
		{attribute 'hide'}
		iOwner						: I_BACnet_ObjectOwner;												// Owner of current Instance (Pointer to current instance per default)
	{endregion}
END_VAR
VAR
	{region 'General'}
		tState						: TCOM_STATE					:= TCOM_STATE.TCOM_STATE_INIT;
		eErrorID					: E_BACnet_Error				:= E_BACnet_Error.eNoError;
		
		tObjectID					: T_BACnet_ObjectIdentifier		:= BACnet_Globals.nBACnetObjId_None;
		
		nCycPropCnt					: DINT;
		nSyncHandlers				: ARRAY [E_BA_SyncMode.eFromSupplement .. E_BA_SyncMode.eToSupplement] OF UDINT;
		bUpdateCOV					: BOOL;
		nPlcSync					: DINT;
		bIsStatic					: BOOL;
	{endregion}
	{region 'Interface Pointer'}
		{attribute 'hide'}
		ipSrv						: ITcIoBACnetPlcServer;
		{attribute 'hide'}
		ipObj						: ITcIoBACnetPlcObject;
	{endregion}
	{region 'Internal'}
		{attribute 'hide'}
		nUpdateCount 				: UDINT := 0;
		{attribute 'conditionalshow'}
		nReqSyncHandlers			: ARRAY [E_BA_SyncMode.eFromSupplement .. E_BA_SyncMode.eToSupplement] OF UDINT;
	{endregion}
END_VAR
VAR PERSISTENT	
	{region 'Internal'}
		{attribute 'conditionalshow'}
		bInitProps					: BOOL	:= TRUE;													// If set, initial property values will be written to BACnet -> in case of reset to origin, values will be rewritten	
	{endregion}			
END_VAR
VAR_STAT
	// (BETA) ... Following symbols should be made non-static / thread safe!
	{region 'Temporary'}
		{attribute 'hide'}
		_fbObjectTmp					: POINTER TO FB_BACnet_Object;
		{attribute 'hide'}
		_fbViewTmp						: POINTER TO FB_BACnet_View;
		{attribute 'hide'}
		_sSymbolPath					: T_MaxString;
		{attribute 'hide'}
		_hResult 						: HRESULT;
		{attribute 'hide'}
		_i								: E_BA_SyncMode;
		{attribute 'hide'}
		_nSize							: DINT;
		{attribute 'hide'}
		_tObjID							: T_BACnet_ObjectIdentifier;
	{endregion}	
END_VAR

// Update device:
IF Server.nUpdateCount = nUpdateCount THEN
	Server();
END_IF
// Remind current number of update counter:
nUpdateCount := Server.nUpdateCount;

IF Server.bOperational THEN
	IF ipObj = 0 THEN
		bReady := FALSE;
		
		IF (iOwner = 0) THEN
			eErrorID := E_BACnet_Error.eInvalidParameter;
			F_BA_LogMessage(ADSLOG_MSGTYPE_ERROR, 'O12', 'Owner of BACnet object not defined!');
		
		ELSIF (NOT Error) THEN
			ipSrv := Server.ServerItf;
			IF ipSrv <> 0 THEN
				IF eObjectType = E_BACnetObjType.ObjDevice THEN
					_hResult := ipSrv.GetObjectByObjectId(ADR(ipObj), 16#23FFFFF);
					IF _hResult = S_OK THEN
						State := TCOM_STATE.TCOM_STATE_PREOP;
					END_IF
				ELSE
					_sSymbolPath := iOwner.SymbolPath;
					_hResult := ipSrv.GetObjectBySymbolName(ADR(ipObj), _sSymbolPath, LEN(_sSymbolPath));
					IF (_hResult = S_OK) THEN
						// Verify existing BACnet-Object type:
						_nSize := SIZEOF(_tObjID);
						IF (S_OK = ipObj.GetPropertyValue(E_BACnetPropIdentifier.PropObjectIdentifier, ADR(_tObjID), ADR(_nSize))) AND_THEN
							(eObjectType <> F_BACnet_GetObjType(_tObjID)) THEN
							// Object type has changed (PLC type differs from stack type)!
							// > Delete existing BACnet-Object:
							ipSrv.DeletePlcObjectRT(ADR(ipObj));
							ipObj := 0;
							
							_hResult := E_FAIL;
						ELSE
							// Continue using existing BACnet-Object:
							bIsStatic := TRUE;			
							State := TCOM_STATE.TCOM_STATE_PREOP;
							
							_hResult := S_OK;
						END_IF
					END_IF
						
					IF (_hResult <> S_OK) THEN
						bInitProps := TRUE;			
						
						// Create new BACnet-Object:
						_hResult := ipSrv.CreatePlcObjectRT(ADR(ipObj), eObjectType, nObjectInstance, TCOM_STATE.TCOM_STATE_PREOP);
						
						IF _hResult = S_OK THEN
							// Init basic properties:
							ipObj.SyncWriteProperty(E_BACnetPropIdentifier.PropPlcSymbolName, ADR(_sSymbolPath), LEN(_sSymbolPath), 16#FFFFFFFF);
					
							State := TCOM_STATE.TCOM_STATE_PREOP;
					
							// Apply requested number of SyncHandlers:
							ApplySyncHandler();
						
							_hResult := ipSrv.CreatePlcObjectRT(ADR(ipObj), eObjectType, nObjectInstance, TCOM_STATE.TCOM_STATE_OP);
							IF _hResult <> S_OK THEN
								eErrorID := E_BACnet_Error.eCreateObject;
								iOwner.LogMsg.Show1(ADSLOG_MSGTYPE_ERROR, 'O37', 'Creating object failed! (Error 0x%x)', F_DINT(_hResult), FALSE);
							END_IF
						ELSE
							eErrorID := E_BACnet_Error.eCreateObject;
							iOwner.LogMsg.Show2(ADSLOG_MSGTYPE_ERROR, 'O46', 'Creating object failed! (Instance: "%d", Error: "0x%x")', F_UDINT(nObjectInstance), F_DINT(_hResult), FALSE);			
						END_IF
					END_IF
				END_IF
			END_IF		
		END_IF	
	ELSE
		IF (Error) THEN
			bReady := FALSE;
		ELSE
			IF (bReady) THEN
				// Instance operational.
				
				// Set number of properties to be synchronized in current cycle:
				nPlcSync := SEL(bUpdateCOV, nCycPropCnt, 255);
			ELSE
				// Complete object initialization:
				State := TCOM_STATE.TCOM_STATE_SAFEOP;
				State := TCOM_STATE.TCOM_STATE_OP;
				
				// Diagnose:
				IF (bInitProps) THEN
					IF (nSyncHandlers[E_BA_SyncMode.eFromSupplement] > nReqSyncHandlers[E_BA_SyncMode.eFromSupplement]) OR
						(nSyncHandlers[E_BA_SyncMode.eToSupplement] > nReqSyncHandlers[E_BA_SyncMode.eToSupplement]) THEN
						iOwner.LogMsg.Show4(ADSLOG_MSGTYPE_WARN, 'O67', 'Inconsistent SyncHandlers! (Requested from/to: %d/%d, Applied from/to: %d/%d)',
											F_UDINT(nReqSyncHandlers[E_BA_SyncMode.eFromSupplement]), F_UDINT(nReqSyncHandlers[E_BA_SyncMode.eToSupplement]),
											F_UDINT(nSyncHandlers[E_BA_SyncMode.eFromSupplement]), F_UDINT(nSyncHandlers[E_BA_SyncMode.eToSupplement]),
											FALSE);	
					END_IF
				END_IF
				
				bReady := NOT Error;
				bInitProps := FALSE;
			END_IF
		END_IF
	END_IF
END_IF

// Unused - Implemented for compatibility reason!
{attribute 'hide'}
METHOD Close
IF ipObj <> 0 THEN
	FW_SafeRelease(ADR(ipObj));
	ipObj:=0;
END_IF

ipSrv := 0;
tState := 0;

FOR _i := E_BA_SyncMode.eFromSupplement TO E_BA_SyncMode.eToSupplement DO
	nSyncHandlers[_i] := 0;
	nReqSyncHandlers[_i] := 0;
END_FOR

bReady := FALSE;
END_METHOD

// Unused - Implemented for compatibility reason!
{attribute 'hide'}
METHOD Execute : BOOL
VAR_INPUT
	bUpdateCOV		: BOOL;
END_VAR
THIS^.bUpdateCOV := bUpdateCOV;

THIS^();

Execute := NOT Error;
END_METHOD

{attribute 'hide'}
METHOD View_RegisterChildObject : BOOL
VAR_INPUT
	iObject			: I_BACnet_BaseObject;
END_VAR
VAR
	_fbObject		: POINTER TO FB_BACnet_BaseObject;
	_sTemp			: T_MaxString;
	_listEntry		: ST_BACnet_DeviceObjectReference;
END_VAR
IF (iObject = 0) THEN
	F_BA_LogMessage(ADSLOG_MSGTYPE_ERROR, 'RCO05', 'Undefined object!');
	
ELSIF (eObjectType <> E_BACnetObjType.ObjStructuredView) THEN
	F_BA_LogMessage(ADSLOG_MSGTYPE_ERROR, 'RCO02', 'Invalid object type!');
	
ELSIF (NOT __QUERYPOINTER(iObject, _fbObject)) THEN
	F_BA_LogMessage(ADSLOG_MSGTYPE_ERROR, 'RCO08', 'Cast of object-interface failed!');
	
ELSE
	_listEntry.objId := iObject.ObjectID;
			
	AddPropertyElementPtr(E_BACnetPropIdentifier.PropSubordinateList, ADR(_listEntry), SIZEOF(_listEntry));

	// (BETA) ... "PropSubordinateAnnotations"
	// > Kann hier das 'ReadPropertyString()' wirklich eingespart werden?? Weil das ja intern UTF8-dekodiert..!?
	(*
	IF (_fbObjectTmp^.ReadPropertyString(E_BACnetPropIdentifier.PropObjectname, _sTemp)) THEN
		AddPropertyElementString(E_BACnetPropIdentifier.PropSubordinateAnnotations, _sTemp);
	END_IF
	*)
	
	// Register child-object in current instance (Called "Subordinate" in BACnet):
	_sTemp := _fbObject^.iOwner.SymbolPath;
	AddPropertyElement(E_BACnetPropIdentifier.PropSubordinateAnnotations, _sTemp);

	View_RegisterChildObject := TRUE;
END_IF
END_METHOD

METHOD PRIVATE DeleteObject : BOOL
IF (ipObj <> 0) AND (ipSrv <> 0) THEN
	IF S_OK <> ipSrv.DeletePlcObjectRT(ADR(ipObj)) THEN
		RETURN;
	END_IF
END_IF 

ipObj := 0;
ipSrv := 0;
eErrorID := E_BACnet_Error.eNoError;

DeleteObject := TRUE;
END_METHOD

METHOD PRIVATE Sched_ReadEntry : BOOL
VAR_INPUT
	eExpectedType	: E_BACnet_ValueChoice;
	pTimeValue		: POINTER TO ST_BACnet_TimeValueList;
END_VAR
VAR_IN_OUT
	entry 			: ST_BA_SchedEntry;
END_VAR
IF (pTimeValue = 0) THEN
	iOwner.LogMsg.Show(ADSLOG_MSGTYPE_WARN, 'SRE02', 'Invalid time value', TRUE);
	
ELSIF (pTimeValue^.stListEntry.stValue.eValueChoice <> E_BACnet_ValueChoice.eNullValue) AND (pTimeValue^.stListEntry.stValue.eValueChoice <> eExpectedType) THEN
	iOwner.LogMsg.Show1(ADSLOG_MSGTYPE_WARN, 'SRE04', 'Invalid time value type "%d"!', F_INT(pTimeValue^.stListEntry.stValue.eValueChoice), TRUE);
	
ELSE
	CASE (pTimeValue^.stListEntry.stValue.eValueChoice) OF
		E_BACnet_ValueChoice.eNullValue:
			entry.eState := E_BA_SchedEntryState.eNull;
			
		E_BACnet_ValueChoice.eEnumerationValue:
			entry.eState := E_BA_SchedEntryState.eValue;
			MEMCPY(ADR(entry.uValue), ADR(pTimeValue^.stListEntry.stValue.stValue.enumValue), pTimeValue^.stListEntry.stValue.nSize - SIZEOF(pTimeValue^.stListEntry.stValue.stValue.choice));
			
	ELSE
		entry.eState := E_BA_SchedEntryState.eValue;
		MEMCPY(ADR(entry.uValue), ADR(pTimeValue^.stListEntry.stValue.stValue), pTimeValue^.stListEntry.stValue.nSize);
	END_CASE
	
	entry.stTime := pTimeValue^.stListEntry.stTime;
	Sched_ReadEntry := TRUE;
END_IF
END_METHOD

METHOD PRIVATE Sched_SetNextDay : BOOL
VAR_IN_OUT
	_pDailySched					: POINTER TO ST_BACnet_DailySchedule;
	_cbTmpSize						: UDINT;
	_cbTotalBuf						: UDINT;
	_pOldTimeValue					: POINTER TO ST_BACnet_TimeValueList;
	_nDayTmp						: DINT;
	_nDayEntryTmp					: DINT;
	_pTimeValue						: POINTER TO ST_BACnet_TimeValueList;
END_VAR
IF eObjectType = E_BACnetObjType.ObjSchedule THEN
	Sched_SetNextDay := ((_pDailySched^.nEntrySize AND 16#80000000) = 16#80000000);
	
	_cbTmpSize := F_BACnet_AlignedSize(_pDailySched^.nEntrySize AND 16#7FFFFFFF) + SIZEOF(_pDailySched^.nEntrySize) + SIZEOF(_pDailySched^.nRes);
	_pDailySched := _pDailySched + _cbTmpSize;
	_cbTotalBuf := _cbTotalBuf + _cbTmpSize;
	_pOldTimeValue := 0;
	_nDayEntryTmp := 1;
	
	IF Sched_SetNextDay THEN
		_pTimeValue := ADR(_pDailySched^.stListEntry);
		_nDayTmp := _nDayTmp + 1;
	END_IF
END_IF
END_METHOD

METHOD PRIVATE Sched_SetNextTimeVal : BOOL
VAR_IN_OUT
	_pDailySched					: POINTER TO ST_BACnet_DailySchedule;
	_pTimeValue						: POINTER TO ST_BACnet_TimeValueList;
	_cbTmpSize						: UDINT;
	_pOldTimeValue					: POINTER TO ST_BACnet_TimeValueList;
END_VAR
IF eObjectType = E_BACnetObjType.ObjSchedule THEN
	Sched_SetNextTimeVal := (_pTimeValue^.nEntrySize AND 16#80000000) = 16#80000000;
	
	_cbTmpSize := F_BACnet_AlignedSize(_pTimeValue^.nEntrySize AND 16#7FFFFFFF) + SIZEOF(_pDailySched^.stListEntry.nEntrySize) + SIZEOF(_pDailySched^.stListEntry.nRes);
	_pOldTimeValue := _pTimeValue;
	_pTimeValue := _pTimeValue + _cbTmpSize;
END_IF
END_METHOD

METHOD PRIVATE Sched_WriteEntry : BOOL
VAR_INPUT
	eValueChoice 	: E_BACnet_ValueChoice;
	pTimeValue		: POINTER TO ST_BACnet_TimeValueList;
	entry 			: ST_BA_SchedEntry;
END_VAR
CASE (entry.eState) OF
	E_BA_SchedEntryState.eNull:
		pTimeValue^.stListEntry.stValue.nSize := 0;
		eValueChoice := E_BACnet_ValueChoice.eNullValue;
		
	E_BA_SchedEntryState.eValue:
		CASE (eValueChoice) OF
			E_BACnet_ValueChoice.eBoolValue:
				pTimeValue^.stListEntry.stValue.nSize := SIZEOF(entry.uValue.bVal);
				
			E_BACnet_ValueChoice.eEnumerationValue:
				pTimeValue^.stListEntry.stValue.nSize := SIZEOF(UDINT) + SIZEOF(E_BACnet_EnumerationValueChoice);
				
			E_BACnet_ValueChoice.eRealValue:
				pTimeValue^.stListEntry.stValue.nSize := SIZEOF(entry.uValue.rVal);
				
			E_BACnet_ValueChoice.eUnsignedValue:
				pTimeValue^.stListEntry.stValue.nSize := SIZEOF(entry.uValue.udiVal);
				
		ELSE
			iOwner.LogMsg.Show(ADSLOG_MSGTYPE_WARN, 'SWE20', 'Unsupported data type!', TRUE);
			RETURN;
		END_CASE
ELSE
	iOwner.LogMsg.Show1(ADSLOG_MSGTYPE_WARN, 'SWE24', 'Unsupported exception scheduler entry type "%d"!', F_INT(entry.eState), TRUE);
	RETURN;
END_CASE
		
// Set data:
pTimeValue^.stListEntry.stTime := entry.stTime;
pTimeValue^.stListEntry.stValue.eValueChoice := eValueChoice;
pTimeValue^.stListEntry.stValue.nRes1 := 0;
IF eValueChoice = E_BACnet_ValueChoice.eEnumerationValue THEN
	pTimeValue^.stListEntry.stValue.stValue.choice := E_BACnet_EnumerationValueChoice.eBinaryPV;
	pTimeValue^.stListEntry.stValue.stValue.enumValue := TO_UDINT(entry.uValue.bVal);
ELSE
	pTimeValue^.stListEntry.stValue.nRes1 := 0;					
	MEMCPY(ADR(pTimeValue^.stListEntry.stValue.stValue), ADR(entry.uValue), pTimeValue^.stListEntry.stValue.nSize);						
END_IF
	
// Calculate time-value entry size:
pTimeValue^.nEntrySize := pTimeValue^.stListEntry.stValue.nSize
						+ SIZEOF(pTimeValue^.stListEntry.nRes)
						+ SIZEOF(pTimeValue^.stListEntry.stTime)
						+ SIZEOF(pTimeValue^.stListEntry.stValue.eValueChoice)
						+ SIZEOF(pTimeValue^.stListEntry.stValue.nRes1)
						+ SIZEOF(pTimeValue^.stListEntry.stValue.nSize);
END_METHOD

METHOD PRIVATE Trend_NextLogRecord : BOOL
VAR_IN_OUT
	_pLbRecordList					: POINTER TO ST_BACnet_LogRecordList;
	_cbTotalBuf						: UDINT;
END_VAR
VAR
	_cbTmpSize						: UDINT;
END_VAR
Trend_NextLogRecord := ((_pLbRecordList^.nEntrySize AND 16#80000000) = 16#80000000);

_cbTmpSize := F_BACnet_AlignedSize(_pLbRecordList^.nEntrySize AND 16#7FFFFFFF) + SIZEOF(_pLbRecordList^.nEntrySize) + SIZEOF(_pLbRecordList^.nSequence);
_pLbRecordList	:= _pLbRecordList + _cbTmpSize;
_cbTotalBuf := _cbTotalBuf + _cbTmpSize;
END_METHOD

METHOD PROTECTED OnObjectStateChanged
CASE (tState) OF
	TCOM_STATE.TCOM_STATE_PREOP:
		// [Hint] To be done in this step:
		// - Disable properties
		// - Initialization of property-memory (e.g. Buffer Size)
		// - Set max. property count via "SetPropertyCount()"
		
		ipObj.GetPropertyValue(E_BACnetPropIdentifier.PropObjectIdentifier, ADR(tObjectID), 0);
		nObjectInstance := F_BACnet_GetObjInstance(tObjectID);
	
		// SyncHandler:
		RequestSyncHandlers(0, 1);
		
	TCOM_STATE.TCOM_STATE_SAFEOP:
		// [Hint] To be done in this step:
		// - Initialize property-sync to important (means COV-indication) properties
		
		SyncProperty(E_BACnetPropIdentifier.PropPlcUpdateTrigger, SIZEOF(nPlcSync), ADR(nPlcSync), 0, eSync_ToSupplement, TRUE);
		
		// Get Object-ID:
		ipObj.GetPropertyValue(E_BACnetPropIdentifier.PropObjectIdentifier, ADR(tObjectID), 0);
		
	TCOM_STATE.TCOM_STATE_OP:
		// [Hint] To be done in this step:
		// - Write protection of properties
		// - Init Entry Count of Arrays: SyncWrite(pData:=Null, nData:=0)
		// - Init Entry Count of Lists: SyncWrite(pData:=ADR(bByteArray), nData:=8)		// -> 'bByteArray' has to be init with NULL
		
		// [Hint] Keep in mind:
		// - Initialize "Resolution" beforce other referring properties are initialized. 
		//   E.g. "COV-Increment"
		// - Register COV-Notification via "SyncProperty(X, Y, Z, bHasChanged, S)":
		//   The trigger variable "bHasChanged" will indicate a COV when if the synchronized property has been written from inside the PLC via "WriteProperty()"-methods.
		
END_CASE

// Notify owner:
iOwner.OnBACnetObjectStateChanged(tState);
END_METHOD

// Called after online change.
{attribute 'call_after_online_change_slot' := '10'}
METHOD PROTECTED OnPostOnlineChange
Close();
END_METHOD

METHOD FB_exit : BOOL
VAR_INPUT
	bInCopyCode : BOOL; // if TRUE, the exit method is called for exiting an instance that is copied afterwards (online change).
END_VAR
Close();
END_METHOD

METHOD Acknowledge : BOOL
VAR_INPUT
	eTransition			: E_BA_EventTransition	:= E_BA_EventTransition.Invalid;
	sMessage			: STRING				:= '';
END_VAR
VAR
	nAckEvent			: UDINT;
END_VAR
IF (Ready) THEN
	CASE (eTransition) OF
		E_BA_EventTransition.eToOffnormal:
			F_BACnet_SetBitFieldBit(ADR(nAckEvent), 2);
		E_BA_EventTransition.eToFault:
			F_BACnet_SetBitFieldBit(ADR(nAckEvent), 1);
		E_BA_EventTransition.eToNormal:
			F_BACnet_SetBitFieldBit(ADR(nAckEvent), 0);
	ELSE
		// Acknowledge all events:
		nAckEvent := 16#FFFFFFFF;
	END_CASE
	
	Acknowledge := (ipObj.SyncAckTransition(TO_UINT(nAckEvent), sMessage, TO_INT(LEN(sMessage))) = S_OK);
END_IF
END_METHOD

PROPERTY Error : BOOL
GET
Error := (eErrorID <> E_BACnet_Error.eNoError);
END_GET
END_PROPERTY

PROPERTY ObjectID : T_BACnet_ObjectIdentifier
GET
ObjectID := tObjectID;
END_GET
END_PROPERTY

PROPERTY ObjectInstance : UDINT
GET
ObjectInstance := nObjectInstance;
END_GET
END_PROPERTY

PROPERTY ObjectType : E_BACnetObjType
GET
ObjectType := eObjectType;
END_GET
END_PROPERTY

PROPERTY Ready : BOOL
GET
Ready := bReady;
END_GET
END_PROPERTY

PROPERTY State : TCOM_STATE
GET
State := tState;
END_GET
SET
PROTECTED
VAR
	_bSetSyncHand	: BOOL;
END_VAR
IF tState <> State THEN
	tState := State;
	OnObjectStateChanged();
END_IF
END_SET
END_PROPERTY

METHOD EnableProperty : HRESULT
VAR_INPUT
	eID : E_BACnetPropIdentifier;
	bEnable : BOOL := TRUE;
END_VAR
EnableProperty := ipObj.SyncPropertyState(eID, bEnable);
END_METHOD

METHOD SetPropertyCount : BOOL
VAR_INPUT
	nCount			: UDINT;
	eSyncMode		: E_BA_SyncMode;
END_VAR
VAR CONSTANT
	LIMIT_MIN		: UDINT		:= 43;
END_VAR
IF (NOT bInitProps) THEN
	// Count already set!
ELSE
	// (BETA) ... SetPropCount
	IF (nCount < LIMIT_MIN) THEN
		nCount := LIMIT_MIN;
	END_IF

	CASE (eSyncMode) OF
		E_BA_SyncMode.eFromSupplement:
			_hResult := WritePropertyUDInt(E_BACnetPropIdentifier.PropCyclicOutMaxCfg, nCount);
		
		E_BA_SyncMode.eToSupplement:
			_hResult := WritePropertyUDInt(E_BACnetPropIdentifier.PropCyclicInMaxCfg, nCount);
			
	ELSE
		iOwner.LogMsg.Show(ADSLOG_MSGTYPE_ERROR, 'SPC23', 'Invalid Sync-Mode defined!', TRUE);
		RETURN;
	END_CASE
	
	IF _hResult = S_OK THEN
		SetPropertyCount := TRUE;
	ELSE
		iOwner.LogMsg.Show1(ADSLOG_MSGTYPE_ERROR, 'SPC20', 'Failed to set property count! (Error 0x%x)', F_DINT(_hResult), TRUE);
	END_IF
END_IF
END_METHOD

METHOD WriteProtectProperty : HRESULT
VAR_INPUT
	eID : E_BACnetPropIdentifier;
	bProtect : BOOL := TRUE;
END_VAR
WriteProtectProperty := ipObj.SyncPropertyProtection(eID, bProtect);
END_METHOD

METHOD AddPropertyElement : BOOL
VAR_INPUT
	eProperty : E_BACnetPropIdentifier;
	xValue : ANY;
END_VAR
VAR
	_stData : POINTER TO ST_BACnet_ValueList;
	_pData : PVOID;
	_nSize : UDINT;
END_VAR
IF (bReady) THEN
	CASE (xValue.TypeClass) OF
		__SYSTEM.TYPE_CLASS.TYPE_STRING:
			AddPropertyElement := (F_BACnet_EncodeUTF8(xValue.pValue, TO_UDINT(xValue.diSize), ADR(BACnet_Globals.stADSBuffer), SIZEOF(BACnet_Globals.stADSBuffer), _nSize) <> 0);
			IF (AddPropertyElement) THEN
				_pData := ADR(BACnet_Globals.stADSBuffer);
			END_IF
			
	ELSE
		iOwner.LogMsg.Show2(ADSLOG_MSGTYPE_ERROR, 'APE10', 'Unimplemented datatype of property "%d"! (Type class "%d")', F_INT(eProperty), F_DWORD(xValue.TypeClass), TRUE);
		RETURN;
	END_CASE
	
	IF (AddPropertyElement) THEN
		_hResult := ipObj.SyncWriteProperty(TO_INT(eProperty), _pData, TO_UINT(F_BACnet_AlignedSize(_nSize)), 16#FFFFFFFE);

		IF (_hResult = S_OK) THEN
			AddPropertyElement := TRUE;
		ELSE
			iOwner.LogMsg.Show2(ADSLOG_MSGTYPE_ERROR, 'APE20', 'Writing element to property "%d" failed! (Error: "0x%x")', F_INT(eProperty), F_DINT(_hResult), TRUE);
		END_IF
	ELSE
		iOwner.LogMsg.Show1(ADSLOG_MSGTYPE_ERROR, 'APE23', 'Failed to prepare element of property "%d"!', F_INT(eProperty), TRUE);
	END_IF
END_IF
END_METHOD

METHOD AddPropertyElementPtr : BOOL
VAR_INPUT
	ePropID : E_BACnetPropIdentifier;
	pData : PVOID;
	nData : UINT;
END_VAR
VAR
	_cbResult : UDINT;
END_VAR
IF (bReady) THEN
	_hResult := ipObj.SyncWriteProperty(TO_INT(ePropID), pData, nData, 16#FFFFFFFE);
	AddPropertyElementPtr:=(S_OK = _hResult);
END_IF
END_METHOD

METHOD RemoveArrayElements : BOOL
VAR_INPUT
	ePropID : E_BACnetPropIdentifier;
END_VAR
_hResult := ipObj.SyncWriteProperty(ePropID, 0, 0, 16#FFFFFFFF);
RemoveArrayElements := (S_OK=_hResult);
END_METHOD

METHOD RemoveListElements : BOOL
VAR_INPUT
	ePropID : E_BACnetPropIdentifier;
END_VAR
VAR
	bData : ARRAY [0 .. 7] OF BYTE;
END_VAR
_hResult := ipObj.SyncWriteProperty(ePropID, ADR(bData), SIZEOF(bData), 16#FFFFFFFF);
RemoveListElements:=(S_OK = _hResult);
END_METHOD

METHOD SetNumberOfStates : BOOL
VAR_INPUT
	nCount			: UDINT;
END_VAR
IF (nCount > 0) THEN
	_hResult := ipObj.SyncWriteProperty(E_BACnetPropIdentifier.PropNumberOfStates, ADR(nCount), SIZEOF(nCount), 16#FFFFFFFF);
	SetNumberOfStates:=(S_OK = _hResult);
END_IF
END_METHOD

METHOD ReadProperty : HRESULT
VAR_INPUT
	ePropID : E_BACnetPropIdentifier;
	pData : PVOID;
	nData : POINTER TO DINT;
END_VAR
VAR
	_size : DINT := 4;
END_VAR
IF (ipObj <> 0) AND (pData <> 0) AND (nData > 0) THEN
	ReadProperty := ipObj.SyncReadProperty(TO_INT(ePropID), pData, nData, 16#FFFFFFFF);

	IF (ReadProperty <> S_OK) THEN
		iOwner.LogMsg.Show2(ADSLOG_MSGTYPE_ERROR, 'RP5', 'Reading property "%d" failed (Error "0x%x")!', F_INT(ePropID), F_DINT(ReadProperty), TRUE);
	END_IF
ELSE
	ReadProperty := E_FAIL;
END_IF
END_METHOD

METHOD ReadPropertyAckedTransitions : HRESULT
VAR CONSTANT
	ePropID : E_BACnetPropIdentifier := E_BACnetPropIdentifier.PropAckedTransitions;
END_VAR

VAR_INPUT
	value : REFERENCE TO ST_BA_EventTransitions;
END_VAR
VAR
	_flags : DWORD;
	_size : DINT := 2;
END_VAR
IF (ipObj <> 0) AND (__ISVALIDREF(value)) THEN
	ReadPropertyAckedTransitions := ipObj.SyncReadProperty(TO_INT(ePropID), ADR(value), ADR(_size), 16#FFFFFFFF);
	
	IF ReadPropertyAckedTransitions = S_OK THEN
		value.bToNormal:= F_BACnet_IsBitFieldBitSet(_flags, E_BACnet_EventTransitionBits.eToNormal);
		value.bToFault:= F_BACnet_IsBitFieldBitSet(_flags, E_BACnet_EventTransitionBits.eToFault);
		value.bToOffnormal:= F_BACnet_IsBitFieldBitSet(_flags, E_BACnet_EventTransitionBits.eToOffnormal);
	END_IF
ELSE
	ReadPropertyAckedTransitions := E_FAIL;
END_IF
END_METHOD

METHOD ReadPropertyBool : HRESULT
VAR_INPUT
	ePropID : E_BACnetPropIdentifier;
	value : REFERENCE TO BOOL;
END_VAR
VAR
	_size : DINT := 1;
END_VAR
IF (ipObj <> 0) AND (__ISVALIDREF(value)) THEN
	ReadPropertyBool := ReadProperty(ePropID, ADR(value), ADR(_size));
ELSE
	ReadPropertyBool := E_FAIL;
END_IF
END_METHOD

METHOD ReadPropertyDateList : HRESULT
VAR_IN_OUT
	stDateList				: ARRAY[*] OF ST_BA_CalendarEntry;
END_VAR
VAR
	_i						: DINT;
	_nLength, _nCount		: DINT;
	_iIndex, _iMin, _iMax	: DINT;
	
	_stEntry				: POINTER TO ST_BACnet_CalendarEntry;
END_VAR
IF (ipObj = 0) THEN
	_hResult := E_FAIL;
ELSE
	_nLength := SIZEOF(BACnet_Globals.bDefaultBuffer);
	_hResult := ReadProperty(E_BACnetPropIdentifier.PropDateList, ADR(BACnet_Globals.bDefaultBuffer), ADR(_nLength));
	
	IF (SUCCEEDED(_hResult)) THEN
		// Clear content:
		MEMSET(stDateList, 0, TO_UDINT(F_BA_DateListSize(stDateList)));
		
		_nCount := (_nLength / SIZEOF(ST_BACnet_CalendarEntry));
		IF (_nCount > 0) THEN
			_iMin := LOWER_BOUND(stDateList, 1);
			_iMax := UPPER_BOUND(stDateList, 1);
			_nCount := MIN(_nCount, (_iMax-_iMin+1));
			
			_stEntry := ADR(BACnet_Globals.bDefaultBuffer);
			_iIndex := _iMin;
			FOR _i := 0 TO (_nCount-1) DO
				stDateList[_iIndex].eType := (_stEntry^.eEventChoice+1);
				stDateList[_iIndex].uDate := (_stEntry^.uCalEntry);
				
				_stEntry := (_stEntry+SIZEOF(ST_BACnet_CalendarEntry));
				_iIndex := (_iIndex+1);
			END_FOR
		END_IF
	END_IF
END_IF

ReadPropertyDateList := _hResult;
END_METHOD

METHOD ReadPropertyEventEnable : HRESULT
VAR CONSTANT
	ePropID : E_BACnetPropIdentifier := E_BACnetPropIdentifier.PropEventEnable;
END_VAR
VAR_INPUT
	value : REFERENCE TO ST_BA_EventTransitions;
END_VAR
VAR
	_flags : WORD := 16#0005;
	_size : DINT := 2;
END_VAR
IF (ipObj <> 0) AND (__ISVALIDREF(value)) THEN
	ReadPropertyEventEnable := ReadProperty(ePropID, ADR(_flags), ADR(_size));
	
	IF (ReadPropertyEventEnable = S_OK) THEN
		value.bToNormal := _flags.13;
		value.bToFault := _flags.14;
		value.bToOffnormal := _flags.15;
	END_IF
ELSE
	ReadPropertyEventEnable := E_FAIL;
END_IF
END_METHOD

METHOD ReadPropertyEventState : HRESULT
VAR CONSTANT
	ePropID : E_BACnetPropIdentifier := E_BACnetPropIdentifier.PropEventState;
END_VAR
VAR_INPUT
	value : REFERENCE TO E_BACnet_EventState;
END_VAR
VAR
	_size : DINT := SIZEOF(E_BACnet_EventState);
END_VAR
IF (ipObj <> 0) AND (__ISVALIDREF(value)) THEN
	ReadPropertyEventState := ReadProperty(ePropID, ADR(value), ADR(_size));
ELSE
	ReadPropertyEventState := E_FAIL;
END_IF
END_METHOD

METHOD ReadPropertyEventTimeStamps : HRESULT
VAR CONSTANT
	ePropID : E_BACnetPropIdentifier := E_BACnetPropIdentifier.PropEventTimeStamps;
END_VAR
VAR_INPUT
	value : REFERENCE TO ST_BACnet_EventTimeStamps;
END_VAR
VAR
	_size : DINT := SIZEOF(ST_BACnet_EventTimeStamps);
END_VAR
IF (ipObj <> 0) AND (__ISVALIDREF(value)) THEN
	ReadPropertyEventTimeStamps := ReadProperty(ePropID, ADR(value), ADR(_size));
ELSE
	ReadPropertyEventTimeStamps := E_FAIL;
END_IF
END_METHOD

METHOD ReadPropertyExceptionSched : HRESULT
VAR_IN_OUT
	tCalendar			: T_BACnet_SchedCalendar;
	tException			: T_BACnet_SchedExceptionList;
END_VAR
VAR_INPUT
	eDatatype			: E_BACnet_ValueChoice;
END_VAR
VAR			
	// General:
	nLenTmp							: UDINT;
	nLength							: DINT;
	
	_cbTmpSize						: UDINT;
	_cbTotalEntry					: UDINT;
	_cbTotalBuf						: UDINT;

	_pDailySched					: POINTER TO ST_BACnet_SpecialEventList;
	_pTimeValue						: POINTER TO ST_BACnet_TimeValueList;
	_nTimeValue						: UDINT;
	_nCalEntry						: UDINT := 1;
	_nExcEntry						: UDINT := 1;
	_calObjId						: T_BACnet_ObjectIdentifier;
END_VAR
IF ipObj = 0 THEN
	_hResult := E_FAIL;	
ELSIF (eDataType = E_BACnet_ValueChoice.eNullValue) THEN
	iOwner.LogMsg.Show(ADSLOG_MSGTYPE_ERROR, 'RWS05', 'Invalid datatype!', TRUE);
	_hResult := E_FAIL;
ELSE
	nLength := SIZEOF(BACnet_Globals.bDefaultBuffer);
	_hResult := ReadProperty(E_BACnetPropIdentifier.PropExceptionSchedule, ADR(BACnet_Globals.bDefaultBuffer), ADR(nLength));
	
	IF (SUCCEEDED(_hResult)) AND (nLength > 8) THEN
		
		// Clear content:
		MEMSET(ADR(tCalendar), 0, SIZEOF(T_BACnet_SchedCalendar));
		MEMSET(ADR(tException), 0, SIZEOF(T_BACnet_SchedExceptionList));
		
		_pDailySched:= ADR(BACnet_Globals.bDefaultBuffer);
		
		WHILE _pDailySched <> 0 DO
			IF _pDailySched^.stEvent.eEventChoice = E_BACnet_SpecialEventChoice.eCalendarReference THEN
				MEMCPY(ADR(_calObjId), ADR(_pDailySched^.stEvent.eCalEntryChoice), SIZEOF(_calObjId));
				tCalendar[_nCalEntry].tRefCalendarID := _calObjId;
				tCalendar[_nCalEntry].eEventPriority := TO_INT(_pDailySched^.stEvent.nEventPriority);
				
